C01819=1084.871,371.355,403.473,176.867,26.567,154.395
C01820=1084.877,371.565,403.441,176.870,26.572,154.396
C01821=1084.882,371.775,403.410,176.873,26.578,154.397
C01822=1084.888,372.022,403.373,176.876,26.584,154.398
C01823=1084.894,372.269,403.336,176.880,26.590,154.399
C01824=1084.900,372.516,403.299,176.883,26.596,154.400
C01825=1084.906,372.763,403.262,176.886,26.603,154.401
C01826=1084.913,373.011,403.225,176.890,26.609,154.403
C01827=1084.919,373.257,403.188,176.892,26.615,154.404
C01828=1084.925,373.504,403.151,176.896,26.621,154.405
C01829=1084.932,373.752,403.115,176.900,26.627,154.406
C01830=1084.937,373.998,403.077,176.902,26.633,154.407
C01831=1084.943,374.246,403.040,176.906,26.640,154.408
C01832=1084.949,374.493,403.003,176.909,26.646,154.409
C01833=1084.956,374.740,402.965,176.913,26.652,154.410
C01834=1084.962,374.988,402.928,176.916,26.658,154.412
C01835=1084.968,375.234,402.891,176.919,26.665,154.413
C01836=1084.974,375.481,402.854,176.923,26.672,154.414
C01837=1084.980,375.728,402.816,176.925,26.678,154.415
C01838=1084.986,375.975,402.780,176.929,26.684,154.416
C01839=1084.993,376.223,402.742,176.933,26.690,154.417
C01840=1084.998,376.469,402.704,176.936,26.697,154.418
C01841=1085.004,376.717,402.667,176.939,26.703,154.420
C01842=1085.011,376.963,402.630,176.942,26.709,154.421
C01843=1085.016,377.210,402.593,176.946,26.716,154.422
C01844=1085.023,377.458,402.555,176.948,26.722,154.423
C01845=1085.029,377.705,402.517,176.952,26.729,154.424
C01846=1085.035,377.952,402.480,176.955,26.736,154.426
C01847=1085.041,378.198,402.443,176.959,26.742,154.427
C01848=1085.047,378.446,402.405,176.962,26.748,154.428
C01849=1085.053,378.693,402.367,176.965,26.755,154.429
C01850=1085.060,378.940,402.330,176.969,26.761,154.430
C01851=1085.066,379.187,402.292,176.972,26.768,154.431
C01852=1085.072,379.434,402.255,176.976,26.775,154.433
C01853=1085.078,379.681,402.217,176.979,26.781,154.434
C01854=1085.084,379.928,402.179,176.982,26.788,154.435
C01855=1085.091,380.174,402.141,176.986,26.795,154.436
C01856=1085.097,380.422,402.104,176.989,26.801,154.438
C01857=1085.103,380.669,402.066,176.993,26.808,154.439
C01858=1085.109,380.916,402.029,176.995,26.814,154.440
C01859=1085.115,381.163,401.991,176.999,26.821,154.441
C01860=1085.122,381.410,401.953,177.002,26.828,154.443
C01861=1085.128,381.657,401.916,177.006,26.834,154.444
C01862=1085.135,381.904,401.877,177.009,26.841,154.445
C01863=1085.141,382.151,401.840,177.012,26.847,154.446
C01864=1085.147,382.398,401.802,177.016,26.854,154.447
C01865=1085.153,382.645,401.764,177.019,26.861,154.449
C01866=1085.159,382.891,401.725,177.022,26.868,154.450
C01867=1085.165,383.138,401.688,177.026,26.875,154.451
C01868=1085.172,383.385,401.649,177.030,26.882,154.453
C01869=1085.178,383.632,401.612,177.032,26.888,154.454
C01870=1085.182,383.856,401.577,177.036,26.895,154.455
C01871=1085.188,384.080,401.542,177.038,26.901,154.456
C01872=1085.194,384.304,401.508,177.042,26.908,154.457
C01873=1085.199,384.527,401.473,177.045,26.914,154.459
C01874=1085.205,384.752,401.438,177.047,26.920,154.460
C01875=1085.211,384.975,401.404,177.051,26.926,154.461
C01876=1085.217,385.199,401.369,177.054,26.932,154.462
C01877=1085.222,385.423,401.334,177.057,26.939,154.463
C01878=1085.228,385.671,401.296,177.061,26.946,154.465
C01879=1085.234,385.917,401.258,177.063,26.953,154.466
C01880=1085.241,386.164,401.220,177.067,26.960,154.467
C01881=1085.247,386.410,401.181,177.070,26.967,154.469
C01882=1085.254,386.658,401.143,177.074,26.974,154.470
C01883=1085.260,386.904,401.105,177.077,26.981,154.471
C01884=1085.266,387.152,401.066,177.081,26.988,154.473
C01885=1085.271,387.399,401.028,177.084,26.995,154.474
C01886=1085.278,387.645,400.989,177.088,27.003,154.475
C01887=1085.284,387.891,400.951,177.091,27.010,154.477
C01888=1085.291,388.139,400.913,177.095,27.017,154.478
C01889=1085.296,388.385,400.874,177.098,27.024,154.479
C01890=1085.303,388.633,400.835,177.101,27.031,154.481
C01891=1085.310,388.880,400.797,177.105,27.038,154.482
C01892=1085.316,389.126,400.758,177.108,27.045,154.484
C01893=1085.322,389.373,400.720,177.111,27.053,154.485
C01894=1085.328,389.620,400.681,177.114,27.060,154.486
C01895=1085.335,389.866,400.642,177.118,27.067,154.488
C01896=1085.341,390.114,400.604,177.121,27.075,154.489
C01897=1085.347,390.360,400.566,177.125,27.082,154.491
C01898=1085.354,390.607,400.526,177.128,27.089,154.492
C01899=1085.360,390.854,400.487,177.132,27.096,154.493
C01900=1085.367,391.100,400.449,177.135,27.104,154.495
C01901=1085.372,391.348,400.410,177.139,27.111,154.496
C01902=1085.379,391.595,400.371,177.142,27.119,154.498
C01903=1085.386,391.841,400.332,177.146,27.126,154.499
C01904=1085.391,392.088,400.293,177.149,27.133,154.500
C01905=1085.398,392.335,400.254,177.152,27.141,154.502
C01906=1085.404,392.582,400.215,177.156,27.148,154.503
C01907=1085.411,392.828,400.177,177.159,27.156,154.505
C01908=1085.417,393.075,400.137,177.163,27.163,154.506
C01909=1085.423,393.322,400.098,177.166,27.171,154.508
C01910=1085.429,393.569,400.059,177.170,27.179,154.509
C01911=1085.436,393.815,400.020,177.173,27.186,154.511
C01912=1085.442,394.062,399.981,177.176,27.194,154.512
C01913=1085.449,394.309,399.942,177.180,27.201,154.514
C01914=1085.455,394.556,399.903,177.183,27.209,154.515
C01915=1085.461,394.803,399.864,177.187,27.217,154.517
C01916=1085.467,395.049,399.824,177.191,27.225,154.518
C01917=1085.474,395.296,399.785,177.194,27.232,154.520
C01918=1085.480,395.543,399.746,177.198,27.240,154.521
C01919=1085.486,395.790,399.706,177.201,27.248,154.523
C01920=1085.493,396.037,399.668,177.205,27.256,154.524
C01921=1085.499,396.283,399.627,177.208,27.264,154.526
C01922=1085.505,396.530,399.588,177.211,27.271,154.527
C01923=1085.511,396.777,399.549,177.215,27.279,154.529
C01924=1085.518,397.023,399.509,177.218,27.287,154.530
C01925=1085.524,397.270,399.470,177.222,27.295,154.532
C01926=1085.530,397.501,399.434,177.225,27.302,154.533
C01927=1085.536,397.732,399.396,177.229,27.310,154.535
C01928=1085.542,397.963,399.360,177.231,27.317,154.536
C01929=1085.548,398.194,399.322,177.235,27.325,154.538
C01930=1085.554,398.424,399.285,177.238,27.332,154.539
C01931=1085.560,398.655,399.248,177.242,27.339,154.541
C01932=1085.566,398.886,399.211,177.245,27.347,154.542
C01933=1085.572,399.116,399.174,177.248,27.354,154.544
C01934=1085.578,399.363,399.134,177.252,27.363,154.545
C01935=1085.585,399.610,399.095,177.255,27.371,154.547
C01936=1085.591,399.856,399.055,177.258,27.379,154.549
C01937=1085.597,400.103,399.015,177.262,27.387,154.550
C01938=1085.604,400.350,398.975,177.265,27.395,154.552
C01939=1085.610,400.596,398.935,177.269,27.404,154.553
C01940=1085.616,400.844,398.896,177.272,27.411,154.555
C01941=1085.622,401.090,398.855,177.276,27.420,154.557
C01942=1085.629,401.337,398.815,177.280,27.428,154.558
C01943=1085.635,401.584,398.776,177.283,27.437,154.560
C01944=1085.641,401.830,398.736,177.286,27.445,154.562
C01945=1085.648,402.077,398.695,177.290,27.453,154.563
C01946=1085.655,402.324,398.655,177.294,27.462,154.565
C01947=1085.661,402.571,398.615,177.297,27.470,154.567
C01948=1085.667,402.817,398.575,177.301,27.478,154.568
C01949=1085.673,403.064,398.535,177.304,27.487,154.570
C01950=1085.680,403.311,398.495,177.308,27.495,154.572
C01951=1085.686,403.557,398.455,177.312,27.504,154.573
C01952=1085.693,403.804,398.415,177.315,27.512,154.575
C01953=1085.700,404.051,398.374,177.318,27.521,154.577
C01954=1085.706,404.297,398.334,177.323,27.529,154.579
C01955=1085.712,404.544,398.294,177.326,27.537,154.580
C01956=1085.719,404.790,398.254,177.329,27.546,154.582
C01957=1085.725,405.037,398.214,177.333,27.555,154.584
C01958=1085.731,405.283,398.174,177.337,27.564,154.586
C01959=1085.738,405.531,398.133,177.340,27.572,154.587
C01960=1085.745,405.777,398.092,177.343,27.581,154.589
C01961=1085.751,406.023,398.051,177.348,27.590,154.591
C01962=1085.757,406.270,398.011,177.351,27.598,154.593
C01963=1085.764,406.517,397.971,177.354,27.607,154.594
C01964=1085.771,406.764,397.931,177.359,27.616,154.596
C01965=1085.776,407.010,397.889,177.362,27.625,154.598
C01966=1085.783,407.256,397.849,177.365,27.634,154.600
C01967=1085.790,407.504,397.809,177.369,27.643,154.602
C01968=1085.797,407.750,397.768,177.373,27.652,154.604
C01969=1085.802,407.996,397.727,177.376,27.660,154.605
C01970=1085.809,408.244,397.686,177.380,27.669,154.607
C01971=1085.815,408.490,397.645,177.383,27.679,154.609
C01972=1085.821,408.736,397.605,177.388,27.688,154.611
C01973=1085.828,408.982,397.564,177.391,27.697,154.613
C01974=1085.834,409.230,397.523,177.394,27.705,154.615
C01975=1085.841,409.476,397.482,177.399,27.715,154.616
C01976=1085.847,409.722,397.441,177.402,27.724,154.618
C01977=1085.854,409.969,397.400,177.406,27.733,154.620
C01978=1085.860,410.216,397.360,177.409,27.742,154.622
C01979=1085.867,410.462,397.318,177.413,27.751,154.624
C01980=1085.874,410.708,397.277,177.417,27.761,154.626
C01981=1085.879,410.955,397.236,177.420,27.770,154.628
C01982=1085.886,411.187,397.198,177.424,27.779,154.630
C01983=1085.892,411.418,397.159,177.428,27.788,154.631
C01984=1085.898,411.649,397.121,177.431,27.796,154.633
C01985=1085.904,411.882,397.082,177.434,27.805,154.635
C01986=1085.910,412.113,397.044,177.438,27.814,154.637
C01987=1085.917,412.344,397.004,177.441,27.822,154.639
C01988=1085.923,412.576,396.965,177.444,27.832,154.641
C01989=1085.929,412.807,396.928,177.449,27.841,154.642
C01990=1085.935,413.054,396.886,177.452,27.850,154.644
C01991=1085.942,413.300,396.845,177.456,27.859,154.646
C01992=1085.948,413.547,396.803,177.459,27.869,154.648
C01993=1085.956,413.793,396.762,177.464,27.878,154.650
C01994=1085.962,414.040,396.720,177.467,27.888,154.652
C01995=1085.969,414.286,396.679,177.471,27.897,154.654
C01996=1085.975,414.532,396.638,177.475,27.907,154.656
C01997=1085.982,414.779,396.596,177.479,27.917,154.658
C01998=1085.988,415.025,396.555,177.483,27.926,154.660
C01999=1085.995,415.272,396.513,177.486,27.936,154.662
C02000=1086.002,415.519,396.472,177.490,27.946,154.664
C02001=1086.008,415.765,396.430,177.494,27.956,154.666
C02002=1086.015,416.011,396.389,177.498,27.966,154.668
C02003=1086.022,416.258,396.347,177.502,27.976,154.671
C02004=1086.028,416.504,396.305,177.505,27.985,154.673
C02005=1086.035,416.751,396.263,177.509,27.996,154.675
C02006=1086.041,416.997,396.221,177.513,28.005,154.677
C02007=1086.048,417.243,396.180,177.517,28.016,154.679
C02008=1086.055,417.490,396.138,177.521,28.025,154.681
C02009=1086.061,417.736,396.096,177.525,28.036,154.683
C02010=1086.067,417.983,396.054,177.529,28.046,154.685
C02011=1086.074,418.229,396.012,177.532,28.056,154.687
C02012=1086.080,418.475,395.970,177.536,28.066,154.690
C02013=1086.087,418.721,395.928,177.541,28.076,154.692
C02014=1086.094,418.968,395.886,177.544,28.086,154.694
C02015=1086.101,419.214,395.844,177.548,28.097,154.696
C02016=1086.107,419.460,395.802,177.552,28.107,154.698
C02017=1086.114,419.707,395.760,177.556,28.117,154.700
C02018=1086.121,419.954,395.718,177.560,28.127,154.703
C02019=1086.127,420.200,395.676,177.564,28.138,154.705
C02020=1086.134,420.445,395.633,177.568,28.149,154.707
C02021=1086.140,420.692,395.592,177.572,28.159,154.709
C02022=1086.147,420.939,395.549,177.575,28.169,154.711
C02023=1086.154,421.185,395.506,177.579,28.180,154.714
C02024=1086.162,421.431,395.465,177.583,28.190,154.716
C02025=1086.168,421.677,395.422,177.588,28.201,154.718
C02026=1086.174,421.923,395.381,177.592,28.211,154.720
C02027=1086.181,422.170,395.338,177.596,28.222,154.723
C02028=1086.188,422.416,395.295,177.599,28.233,154.725
C02029=1086.194,422.663,395.252,177.603,28.244,154.727
C02030=1086.201,422.909,395.210,177.607,28.254,154.730
C02031=1086.208,423.155,395.167,177.611,28.265,154.732
C02032=1086.215,423.401,395.125,177.616,28.276,154.734
C02033=1086.221,423.647,395.083,177.620,28.287,154.737
C02034=1086.228,423.893,395.040,177.624,28.298,154.739
C02035=1086.234,424.140,394.997,177.627,28.309,154.741
C02036=1086.241,424.386,394.954,177.631,28.319,154.744
C02037=1086.248,424.632,394.911,177.635,28.331,154.746
C02038=1086.259,425.045,394.840,177.642,28.349,154.750
C02039=1086.271,425.458,394.768,177.649,28.368,154.754
C02040=1086.282,425.871,394.696,177.656,28.386,154.758
C02041=1086.293,426.284,394.624,177.663,28.405,154.762
C02042=1086.300,426.529,394.581,177.667,28.417,154.765
C02043=1086.307,426.775,394.538,177.671,28.428,154.767
C02044=1086.313,427.022,394.495,177.675,28.439,154.769
C02045=1086.320,427.268,394.452,177.679,28.450,154.772
C02046=1086.327,427.514,394.409,177.683,28.462,154.774
C02047=1086.334,427.760,394.366,177.687,28.473,154.777
C02048=1086.341,428.006,394.322,177.691,28.485,154.779
C02049=1086.348,428.253,394.279,177.695,28.496,154.782
C02050=1086.356,428.498,394.236,177.700,28.507,154.784
C02051=1086.362,428.745,394.193,177.704,28.519,154.787
C02052=1086.369,428.991,394.149,177.709,28.531,154.789
C02053=1086.375,429.237,394.106,177.713,28.543,154.792
C02054=1086.382,429.482,394.062,177.717,28.555,154.795
C02055=1086.389,429.729,394.019,177.721,28.566,154.797
C02056=1086.396,429.974,393.976,177.725,28.578,154.800
C02057=1086.403,430.221,393.932,177.729,28.590,154.802
C02058=1086.410,430.467,393.888,177.733,28.602,154.805
C02059=1086.416,430.713,393.845,177.737,28.614,154.808
C02060=1086.423,430.958,393.801,177.741,28.626,154.810
C02061=1086.430,431.204,393.757,177.746,28.638,154.813
C02062=1086.437,431.451,393.713,177.751,28.650,154.815
C02063=1086.444,431.697,393.670,177.755,28.662,154.818
C02064=1086.450,431.943,393.626,177.759,28.674,154.821
C02065=1086.458,432.188,393.583,177.763,28.686,154.823
C02066=1086.465,432.435,393.539,177.767,28.698,154.826
C02067=1086.472,432.681,393.495,177.772,28.710,154.829
C02068=1086.478,432.927,393.452,177.776,28.723,154.832
C02069=1086.485,433.173,393.407,177.780,28.735,154.834
C02070=1086.492,433.419,393.363,177.784,28.748,154.837
C02071=1086.499,433.664,393.320,177.789,28.760,154.840
C02072=1086.506,433.911,393.275,177.793,28.773,154.843
C02073=1086.513,434.156,393.231,177.797,28.785,154.845
C02074=1086.521,434.468,393.175,177.803,28.801,154.849
C02075=1086.530,434.780,393.119,177.808,28.817,154.852
C02076=1086.539,435.092,393.063,177.814,28.833,154.856
C02077=1086.548,435.404,393.007,177.820,28.849,154.860
C02078=1086.555,435.649,392.963,177.824,28.862,154.862
C02079=1086.561,435.895,392.919,177.829,28.875,154.865
C02080=1086.569,436.141,392.874,177.833,28.888,154.868
C02081=1086.575,436.387,392.829,177.837,28.901,154.871
C02082=1086.583,436.633,392.786,177.842,28.914,154.874
C02083=1086.590,436.878,392.741,177.846,28.926,154.877
C02084=1086.597,437.124,392.696,177.850,28.939,154.880
C02085=1086.604,437.370,392.651,177.855,28.953,154.883
C02086=1086.611,437.616,392.607,177.859,28.966,154.886
C02087=1086.618,437.862,392.563,177.864,28.979,154.888
C02088=1086.625,438.108,392.518,177.868,28.992,154.891
C02089=1086.632,438.353,392.473,177.872,29.005,154.894
C02090=1086.639,438.584,392.432,177.876,29.018,154.897
C02091=1086.646,438.814,392.390,177.881,29.030,154.900
C02092=1086.652,439.044,392.347,177.886,29.043,154.903
C02093=1086.658,439.274,392.306,177.890,29.056,154.906
C02094=1086.666,439.505,392.263,177.894,29.068,154.909
C02095=1086.672,439.735,392.222,177.898,29.081,154.911
C02096=1086.679,439.966,392.179,177.902,29.093,154.914
C02097=1086.686,440.196,392.137,177.907,29.106,154.917
C02098=1086.693,440.442,392.092,177.911,29.120,154.920
C02099=1086.700,440.687,392.047,177.916,29.134,154.923
C02100=1086.707,440.933,392.002,177.920,29.147,154.926
C02101=1086.715,441.179,391.957,177.925,29.161,154.930
C02102=1086.721,441.424,391.912,177.930,29.175,154.933
C02103=1086.728,441.670,391.867,177.934,29.189,154.936
C02104=1086.736,441.916,391.821,177.939,29.203,154.939
C02105=1086.743,442.162,391.776,177.943,29.217,154.942
C02106=1086.750,442.407,391.732,177.948,29.231,154.945
C02107=1086.756,442.653,391.685,177.952,29.245,154.949
C02108=1086.764,442.898,391.640,177.957,29.260,154.952
C02109=1086.771,443.144,391.595,177.962,29.274,154.955
C02110=1086.778,443.389,391.549,177.966,29.288,154.958
C02111=1086.785,443.635,391.504,177.971,29.302,154.962
C02112=1086.793,443.881,391.458,177.976,29.317,154.965
C02113=1086.800,444.127,391.412,177.980,29.331,154.968
C02114=1086.807,444.373,391.367,177.985,29.346,154.972
C02115=1086.815,444.618,391.321,177.991,29.360,154.975
C02116=1086.821,444.863,391.276,177.995,29.374,154.978
C02117=1086.829,445.109,391.230,178.000,29.389,154.981
C02118=1086.836,445.354,391.184,178.004,29.404,154.985
C02119=1086.843,445.600,391.138,178.008,29.418,154.988
C02120=1086.851,445.845,391.092,178.012,29.433,154.992
C02121=1086.858,446.091,391.046,178.016,29.448,154.995
C02122=1086.865,446.336,391.001,178.019,29.462,154.999
C02123=1086.872,446.582,390.954,178.022,29.477,155.002
C02124=1086.880,446.828,390.909,178.025,29.491,155.005
C02125=1086.887,447.073,390.862,178.029,29.506,155.009
C02126=1086.894,447.319,390.817,178.032,29.520,155.012
C02127=1086.901,447.565,390.771,178.034,29.535,155.016
C02128=1086.908,447.810,390.724,178.036,29.549,155.019
C02129=1086.916,448.056,390.679,178.038,29.563,155.023
C02130=1086.923,448.301,390.632,178.040,29.578,155.027
C02131=1086.931,448.546,390.586,178.043,29.593,155.030
C02132=1086.938,448.793,390.539,178.044,29.607,155.034
C02133=1086.946,449.038,390.494,178.045,29.621,155.037
C02134=1086.952,449.283,390.447,178.046,29.636,155.041
C02135=1086.960,449.527,390.401,178.048,29.650,155.044
C02136=1086.969,449.773,390.355,178.049,29.664,155.048
C02137=1086.980,450.019,390.311,178.050,29.676,155.051
C02138=1086.604,450.011,390.111,178.013,29.864,155.102
C02139=1086.592,449.765,390.155,178.012,29.851,155.098
C02140=1086.583,449.520,390.202,178.010,29.837,155.095
C02141=1086.576,449.275,390.247,178.009,29.823,155.091
C02142=1086.568,449.031,390.293,178.007,29.808,155.088
C02143=1086.561,448.785,390.339,178.006,29.794,155.084
C02144=1086.554,448.540,390.386,178.005,29.780,155.081
C02145=1086.546,448.294,390.432,178.002,29.765,155.077
C02146=1086.539,448.048,390.479,178.000,29.750,155.074
C02147=1086.531,447.803,390.525,177.998,29.736,155.070
C02148=1086.524,447.557,390.571,177.995,29.721,155.066
C02149=1086.516,447.312,390.617,177.993,29.707,155.063
C02150=1086.510,447.066,390.663,177.990,29.693,155.060
C02151=1086.503,446.820,390.709,177.987,29.678,155.056
C02152=1086.495,446.576,390.756,177.983,29.663,155.053
C02153=1086.488,446.330,390.802,177.980,29.649,155.049
C02154=1086.480,446.084,390.848,177.977,29.634,155.046
C02155=1086.473,445.839,390.894,177.973,29.619,155.042
C02156=1086.466,445.593,390.940,177.969,29.605,155.039
C02157=1086.459,445.347,390.986,177.964,29.590,155.035
C02158=1086.451,445.102,391.031,177.960,29.576,155.032
C02159=1086.443,444.857,391.077,177.955,29.561,155.029
C02160=1086.437,444.611,391.123,177.950,29.546,155.025
C02161=1086.429,444.365,391.168,177.946,29.532,155.022
C02162=1086.422,444.119,391.214,177.941,29.517,155.019
C02163=1086.415,443.874,391.260,177.935,29.503,155.015
C02164=1086.407,443.628,391.306,177.931,29.489,155.012
C02165=1086.401,443.383,391.352,177.926,29.474,155.009
C02166=1086.393,443.137,391.397,177.921,29.460,155.005
C02167=1086.386,442.892,391.442,177.917,29.446,155.002
C02168=1086.378,442.646,391.487,177.912,29.431,154.999
C02169=1086.372,442.400,391.533,177.907,29.417,154.996
C02170=1086.365,442.155,391.579,177.902,29.403,154.993
C02171=1086.357,441.909,391.624,177.897,29.389,154.989
C02172=1086.350,441.664,391.669,177.893,29.375,154.986
C02173=1086.343,441.417,391.715,177.888,29.361,154.983
C02174=1086.336,441.172,391.759,177.884,29.347,154.980
C02175=1086.329,440.927,391.805,177.879,29.333,154.977
C02176=1086.321,440.680,391.850,177.874,29.320,154.974
C02177=1086.314,440.434,391.895,177.869,29.306,154.971
C02178=1086.307,440.190,391.940,177.865,29.292,154.967
C02179=1086.301,439.966,391.982,177.861,29.280,154.965
C02180=1086.294,439.742,392.022,177.857,29.267,154.962
C02181=1086.288,439.519,392.063,177.852,29.255,154.959
C02182=1086.281,439.295,392.104,177.848,29.243,154.956
C02183=1086.275,439.072,392.145,177.844,29.231,154.954
C02184=1086.267,438.849,392.185,177.839,29.218,154.951
C02185=1086.261,438.626,392.226,177.836,29.206,154.948
C02186=1086.255,438.402,392.267,177.832,29.194,154.945
C02187=1086.247,438.156,392.312,177.826,29.181,154.942
C02188=1086.241,437.911,392.356,177.822,29.168,154.939
C02189=1086.233,437.665,392.401,177.818,29.155,154.936
C02190=1086.227,437.420,392.446,177.813,29.141,154.933
C02191=1086.220,437.173,392.490,177.809,29.128,154.931
C02192=1086.212,436.927,392.535,177.804,29.115,154.928
C02193=1086.206,436.681,392.579,177.800,29.102,154.925
C02194=1086.199,436.436,392.624,177.795,29.089,154.922
C02195=1086.191,436.190,392.667,177.790,29.076,154.919
C02196=1086.184,435.944,392.712,177.786,29.063,154.916
C02197=1086.177,435.698,392.757,177.782,29.050,154.913
C02198=1086.171,435.452,392.801,177.777,29.037,154.910
C02199=1086.163,435.206,392.846,177.773,29.025,154.907
C02200=1086.157,434.961,392.890,177.768,29.012,154.905
C02201=1086.150,434.714,392.935,177.764,28.999,154.902
C02202=1086.142,434.469,392.979,177.759,28.987,154.899
C02203=1086.136,434.223,393.022,177.755,28.974,154.896
C02204=1086.129,433.977,393.067,177.751,28.961,154.893
C02205=1086.122,433.731,393.111,177.747,28.949,154.891
C02206=1086.115,433.485,393.155,177.742,28.936,154.888
C02207=1086.107,433.240,393.199,177.738,28.924,154.885
C02208=1086.101,432.994,393.243,177.733,28.912,154.882
C02209=1086.095,432.748,393.287,177.729,28.899,154.880
C02210=1086.088,432.501,393.331,177.725,28.887,154.877
C02211=1086.080,432.255,393.374,177.720,28.875,154.874
C02212=1086.074,432.010,393.419,177.716,28.863,154.872
C02213=1086.066,431.764,393.463,177.712,28.851,154.869
C02214=1086.059,431.518,393.507,177.707,28.838,154.866
C02215=1086.052,431.272,393.550,177.703,28.826,154.863
C02216=1086.045,431.025,393.594,177.699,28.815,154.861
C02217=1086.039,430.779,393.638,177.694,28.802,154.858
C02218=1086.032,430.534,393.681,177.690,28.790,154.856
C02219=1086.025,430.288,393.725,177.686,28.778,154.853
C02220=1086.018,430.042,393.768,177.681,28.766,154.850
C02221=1086.011,429.795,393.812,177.677,28.755,154.848
C02222=1086.004,429.550,393.856,177.673,28.743,154.845
C02223=1085.998,429.303,393.899,177.669,28.731,154.843
C02224=1085.991,429.057,393.942,177.665,28.720,154.840
C02225=1085.984,428.811,393.986,177.661,28.708,154.838
C02226=1085.977,428.566,394.029,177.656,28.696,154.835
C02227=1085.970,428.318,394.073,177.652,28.685,154.832
C02228=1085.963,428.073,394.116,177.648,28.673,154.830
C02229=1085.956,427.827,394.159,177.643,28.661,154.827
C02230=1085.949,427.581,394.202,177.639,28.650,154.825
C02231=1085.943,427.335,394.246,177.634,28.639,154.822
C02232=1085.936,427.089,394.288,177.630,28.627,154.820
C02233=1085.929,426.843,394.331,177.626,28.616,154.817
C02234=1085.922,426.596,394.375,177.622,28.604,154.815
C02235=1085.915,426.356,394.417,177.619,28.593,154.813
C02236=1085.908,426.116,394.458,177.614,28.582,154.810
C02237=1085.902,425.877,394.501,177.610,28.571,154.808
C02238=1085.896,425.636,394.542,177.606,28.561,154.806
C02239=1085.889,425.397,394.585,177.602,28.549,154.803
C02240=1085.882,425.157,394.626,177.598,28.539,154.801
C02241=1085.876,424.917,394.667,177.594,28.528,154.799
C02242=1085.869,424.677,394.710,177.590,28.517,154.796
C02243=1085.862,424.431,394.752,177.586,28.506,154.794
C02244=1085.855,424.184,394.795,177.582,28.495,154.791
C02245=1085.849,423.938,394.837,177.577,28.484,154.789
C02246=1085.842,423.692,394.881,177.574,28.473,154.787
C02247=1085.835,423.446,394.924,177.570,28.462,154.784
C02248=1085.828,423.200,394.966,177.566,28.452,154.782
C02249=1085.822,422.953,395.009,177.562,28.441,154.780
C02250=1085.815,422.707,395.051,177.557,28.430,154.777
C02251=1085.808,422.461,395.094,177.553,28.419,154.775
C02252=1085.802,422.215,395.137,177.549,28.408,154.773
C02253=1085.796,421.969,395.179,177.546,28.398,154.771
C02254=1085.789,421.722,395.222,177.542,28.387,154.768
C02255=1085.781,421.476,395.263,177.537,28.376,154.766
C02256=1085.775,421.229,395.306,177.533,28.366,154.764
C02257=1085.768,420.983,395.348,177.529,28.355,154.761
C02258=1085.761,420.737,395.391,177.526,28.345,154.759
C02259=1085.754,420.491,395.433,177.522,28.334,154.757
C02260=1085.748,420.244,395.475,177.517,28.324,154.755
C02261=1085.741,419.998,395.517,177.513,28.314,154.753
C02262=1085.734,419.752,395.560,177.510,28.303,154.750
C02263=1085.724,419.343,395.630,177.503,28.286,154.747
C02264=1085.712,418.933,395.699,177.497,28.269,154.743
C02265=1085.702,418.525,395.769,177.490,28.252,154.740
C02266=1085.690,418.115,395.839,177.484,28.235,154.736
C02267=1085.684,417.869,395.881,177.479,28.225,154.734
C02268=1085.677,417.623,395.923,177.475,28.215,154.732
C02269=1085.670,417.376,395.965,177.472,28.205,154.730
C02270=1085.664,417.130,396.007,177.467,28.195,154.727
C02271=1085.657,416.884,396.049,177.463,28.184,154.725
C02272=1085.650,416.637,396.090,177.460,28.175,154.723
C02273=1085.644,416.391,396.132,177.456,28.164,154.721
C02274=1085.637,416.144,396.174,177.452,28.154,154.719
C02275=1085.631,415.898,396.216,177.448,28.145,154.717
C02276=1085.624,415.652,396.257,177.444,28.135,154.715
C02277=1085.618,415.405,396.299,177.441,28.125,154.713
C02278=1085.610,415.159,396.341,177.436,28.115,154.711
C02279=1085.604,414.913,396.382,177.432,28.106,154.709
C02280=1085.597,414.666,396.424,177.429,28.096,154.707
C02281=1085.591,414.420,396.465,177.425,28.086,154.705
C02282=1085.584,414.173,396.507,177.421,28.077,154.703
C02283=1085.577,413.926,396.548,177.417,28.067,154.701
C02284=1085.571,413.680,396.590,177.414,28.058,154.699
C02285=1085.564,413.434,396.631,177.409,28.048,154.697
C02286=1085.558,413.187,396.672,177.406,28.039,154.695
C02287=1085.551,412.941,396.714,177.402,28.029,154.693
C02288=1085.545,412.695,396.755,177.399,28.020,154.691
C02289=1085.537,412.448,396.796,177.394,28.010,154.689
C02290=1085.531,412.202,396.838,177.391,28.000,154.687
C02291=1085.523,411.900,396.888,177.386,27.989,154.684
C02292=1085.515,411.598,396.938,177.381,27.978,154.682
C02293=1085.506,411.297,396.989,177.376,27.966,154.680
C02294=1085.500,410.996,397.039,177.372,27.955,154.677
C02295=1085.492,410.749,397.080,177.368,27.945,154.676
C02296=1085.487,410.502,397.121,177.365,27.936,154.674
C02297=1085.479,410.256,397.162,177.360,27.927,154.672
C02298=1085.473,410.010,397.203,177.357,27.918,154.670
C02299=1085.467,409.763,397.244,177.354,27.908,154.668
C02300=1085.460,409.517,397.285,177.349,27.899,154.666
C02301=1085.454,409.270,397.326,177.346,27.890,154.664
C02302=1085.447,409.023,397.367,177.342,27.881,154.662
C02303=1085.440,408.777,397.408,177.339,27.872,154.660
C02304=1085.435,408.530,397.448,177.335,27.863,154.658
C02305=1085.428,408.283,397.489,177.331,27.854,154.657
C02306=1085.422,408.037,397.530,177.328,27.845,154.655
C02307=1085.415,407.790,397.571,177.324,27.836,154.653
C02308=1085.409,407.545,397.611,177.320,27.827,154.651
C02309=1085.402,407.297,397.653,177.317,27.818,154.649
C02310=1085.396,407.051,397.693,177.312,27.809,154.647
C02311=1085.389,406.805,397.734,177.309,27.800,154.646
C02312=1085.382,406.557,397.774,177.306,27.791,154.644
C02313=1085.377,406.311,397.815,177.302,27.782,154.642
C02314=1085.370,406.065,397.856,177.298,27.774,154.640
C02315=1085.364,405.818,397.896,177.295,27.765,154.638
C02316=1085.357,405.571,397.936,177.291,27.756,154.637
C02317=1085.350,405.324,397.976,177.287,27.747,154.635
C02318=1085.345,405.078,398.017,177.284,27.739,154.633
C02319=1085.338,404.831,398.057,177.280,27.730,154.631
C02320=1085.331,404.584,398.098,177.277,27.722,154.630
C02321=1085.325,404.337,398.138,177.272,27.713,154.628
C02322=1085.318,404.091,398.179,177.269,27.704,154.626
C02323=1085.312,403.845,398.219,177.266,27.696,154.624
C02324=1085.305,403.598,398.259,177.262,27.687,154.623
C02325=1085.299,403.352,398.299,177.258,27.679,154.621
C02326=1085.292,403.104,398.339,177.255,27.670,154.619
C02327=1085.286,402.858,398.379,177.251,27.662,154.618
C02328=1085.280,402.611,398.419,177.248,27.654,154.616
C02329=1085.273,402.365,398.460,177.243,27.645,154.614
C02330=1085.267,402.118,398.500,177.240,27.636,154.612
C02331=1085.260,401.872,398.540,177.237,27.628,154.611
C02332=1085.254,401.625,398.580,177.233,27.620,154.609
C02333=1085.247,401.377,398.620,177.230,27.612,154.607
C02334=1085.241,401.131,398.660,177.226,27.604,154.606
C02335=1085.235,400.884,398.700,177.222,27.595,154.604
C02336=1085.228,400.638,398.740,177.219,27.587,154.603
C02337=1085.222,400.390,398.780,177.215,27.579,154.601
C02338=1085.216,400.144,398.820,177.212,27.570,154.599
C02339=1085.209,399.897,398.860,177.208,27.562,154.598
C02340=1085.203,399.651,398.899,177.205,27.554,154.596
C02341=1085.196,399.404,398.939,177.201,27.545,154.594
C02342=1085.190,399.158,398.979,177.197,27.538,154.593
C02343=1085.184,398.926,399.016,177.195,27.530,154.591
C02344=1085.178,398.694,399.053,177.191,27.523,154.590
C02345=1085.172,398.464,399.090,177.188,27.515,154.588
C02346=1085.166,398.233,399.128,177.184,27.508,154.587
C02347=1085.160,398.001,399.165,177.181,27.500,154.585
C02348=1085.154,397.769,399.201,177.178,27.493,154.584
C02349=1085.148,397.538,399.239,177.175,27.485,154.582
C02350=1085.143,397.307,399.276,177.171,27.478,154.581
C02351=1085.136,397.061,399.315,177.168,27.470,154.579
C02352=1085.129,396.814,399.355,177.164,27.462,154.578
C02353=1085.123,396.567,399.394,177.161,27.454,154.576
C02354=1085.117,396.320,399.434,177.157,27.446,154.575
C02355=1085.110,396.074,399.473,177.154,27.438,154.573
C02356=1085.104,395.826,399.513,177.150,27.431,154.572
C02357=1085.098,395.579,399.552,177.147,27.423,154.570
C02358=1085.091,395.333,399.591,177.144,27.415,154.568
C02359=1085.085,395.087,399.631,177.140,27.407,154.567
C02360=1085.079,394.840,399.670,177.137,27.400,154.565
C02361=1085.073,394.593,399.709,177.133,27.392,154.564
C02362=1085.067,394.346,399.749,177.130,27.384,154.562
C02363=1085.060,394.099,399.788,177.126,27.377,154.561
C02364=1085.054,393.852,399.827,177.122,27.368,154.559
C02365=1085.047,393.606,399.865,177.118,27.361,154.558
C02366=1085.041,393.358,399.905,177.115,27.354,154.557
C02367=1085.035,393.112,399.944,177.111,27.346,154.555
C02368=1085.028,392.865,399.984,177.108,27.338,154.554
C02369=1085.022,392.619,400.022,177.105,27.330,154.552
C02370=1085.016,392.372,400.062,177.101,27.323,154.551
C02371=1085.009,392.124,400.100,177.097,27.316,154.549
C02372=1085.004,391.878,400.139,177.095,27.308,154.548
C02373=1084.997,391.631,400.178,177.092,27.301,154.546
C02374=1084.990,391.384,400.217,177.088,27.293,154.545
C02375=1084.984,391.137,400.256,177.085,27.286,154.543
C02376=1084.978,390.891,400.294,177.081,27.279,154.542
C02377=1084.971,390.644,400.333,177.078,27.271,154.540
C02378=1084.965,390.397,400.373,177.074,27.264,154.539
C02379=1084.959,390.150,400.411,177.070,27.257,154.538
C02380=1084.952,389.903,400.449,177.067,27.249,154.536
C02381=1084.946,389.657,400.488,177.064,27.242,154.535
C02382=1084.940,389.410,400.527,177.060,27.235,154.534
C02383=1084.934,389.163,400.565,177.057,27.227,154.532
C02384=1084.927,388.916,400.604,177.053,27.220,154.531
C02385=1084.921,388.670,400.643,177.049,27.213,154.529
C02386=1084.914,388.422,400.681,177.046,27.206,154.528
C02387=1084.908,388.175,400.720,177.042,27.199,154.527
C02388=1084.902,387.929,400.759,177.039,27.191,154.525
C02389=1084.895,387.682,400.797,177.035,27.184,154.524
C02390=1084.889,387.436,400.835,177.032,27.177,154.523
C02391=1084.883,387.188,400.873,177.028,27.170,154.521
C02392=1084.877,386.942,400.912,177.026,27.163,154.520
C02393=1084.871,386.694,400.951,177.022,27.156,154.518
C02394=1084.864,386.448,400.989,177.019,27.149,154.517
C02395=1084.858,386.201,401.027,177.015,27.142,154.516
C02396=1084.851,385.954,401.066,177.012,27.135,154.514
C02397=1084.845,385.707,401.104,177.008,27.128,154.513
C02398=1084.840,385.461,401.143,177.005,27.120,154.512
C02399=1084.834,385.236,401.177,177.002,27.114,154.511
C02400=1084.828,385.012,401.212,176.998,27.108,154.509
C02401=1084.823,384.787,401.247,176.996,27.101,154.508
C02402=1084.816,384.563,401.282,176.993,27.095,154.507
C02403=1084.811,384.337,401.316,176.989,27.089,154.506
C02404=1084.806,384.114,401.351,176.987,27.082,154.505
C02405=1084.800,383.890,401.386,176.983,27.076,154.503
C02406=1084.794,383.665,401.420,176.980,27.070,154.502
C02407=1084.789,383.418,401.459,176.977,27.063,154.501
C02408=1084.782,383.171,401.497,176.973,27.056,154.500
C02409=1084.776,382.924,401.534,176.971,27.049,154.498
C02410=1084.770,382.677,401.572,176.967,27.042,154.497
C02411=1084.764,382.431,401.611,176.963,27.036,154.496
C02412=1084.758,382.184,401.649,176.960,27.029,154.495
C02413=1084.751,381.936,401.687,176.956,27.022,154.493
C02414=1084.745,381.690,401.725,176.953,27.015,154.492
C02415=1084.738,381.442,401.762,176.950,27.009,154.491
C02416=1084.732,381.196,401.800,176.947,27.002,154.489
C02417=1084.726,380.949,401.838,176.943,26.995,154.488
C02418=1084.720,380.702,401.876,176.939,26.988,154.487
C02419=1084.714,380.455,401.914,176.937,26.982,154.486
C02420=1084.707,380.207,401.952,176.933,26.975,154.485
C02421=1084.701,379.961,401.989,176.930,26.969,154.483
C02422=1084.695,379.714,402.026,176.926,26.962,154.482
C02423=1084.689,379.466,402.064,176.923,26.955,154.481
C02424=1084.683,379.219,402.102,176.920,26.949,154.480
C02425=1084.677,378.973,402.140,176.916,26.942,154.479
C02426=1084.670,378.726,402.177,176.913,26.936,154.477
C02427=1084.664,378.479,402.215,176.909,26.929,154.476
C02428=1084.658,378.231,402.252,176.906,26.923,154.475
C02429=1084.652,377.985,402.290,176.903,26.916,154.474
C02430=1084.646,377.737,402.328,176.899,26.909,154.472
C02431=1084.639,377.491,402.365,176.896,26.903,154.471
C02432=1084.633,377.243,402.402,176.893,26.897,154.470
C02433=1084.627,376.997,402.440,176.889,26.890,154.469
C02434=1084.621,376.749,402.478,176.886,26.884,154.468
C02435=1084.615,376.502,402.514,176.883,26.878,154.467
C02436=1084.609,376.255,402.552,176.880,26.871,154.465
C02437=1084.603,376.008,402.589,176.876,26.865,154.464
C02438=1084.596,375.762,402.626,176.872,26.858,154.463
C02439=1084.590,375.514,402.664,176.870,26.852,154.462
C02440=1084.584,375.267,402.701,176.866,26.845,154.461
C02441=1084.578,375.020,402.739,176.863,26.839,154.460
C02442=1084.572,374.773,402.776,176.860,26.833,154.458
C02443=1084.566,374.526,402.813,176.856,26.826,154.457
C02444=1084.561,374.279,402.850,176.853,26.820,154.456
C02445=1084.554,374.031,402.887,176.850,26.814,154.455
C02446=1084.548,373.784,402.925,176.846,26.807,154.454
C02447=1084.541,373.537,402.961,176.843,26.801,154.453
C02448=1084.536,373.290,402.998,176.840,26.795,154.452
C02449=1084.529,373.044,403.036,176.836,26.789,154.450
C02450=1084.524,372.796,403.073,176.833,26.783,154.449
C02451=1084.517,372.548,403.109,176.830,26.776,154.448
C02452=1084.511,372.302,403.147,176.826,26.770,154.447
C02453=1084.504,372.055,403.184,176.823,26.764,154.446
C02454=1084.498,371.808,403.220,176.820,26.758,154.445
C02455=1084.494,371.597,403.252,176.817,26.753,154.444
C02456=1084.488,371.386,403.283,176.814,26.748,154.443
C02457=1084.483,371.176,403.314,176.812,26.742,154.442
C02458=1084.477,370.967,403.346,176.809,26.737,154.441
C02459=1084.471,370.756,403.378,176.806,26.732,154.440
C02460=1084.467,370.546,403.409,176.803,26.727,154.439
C02461=1084.462,370.336,403.440,176.800,26.722,154.438
C02462=1084.456,370.125,403.472,176.797,26.716,154.438
C02463=1084.450,369.878,403.508,176.794,26.710,154.437
C02464=1084.444,369.630,403.545,176.791,26.705,154.435
C02465=1084.438,369.383,403.582,176.787,26.699,154.434
C02466=1084.432,369.136,403.618,176.785,26.692,154.433
C02467=1084.426,368.889,403.655,176.781,26.686,154.432
C02468=1084.420,368.642,403.692,176.777,26.680,154.431
C02469=1084.414,368.395,403.729,176.775,26.674,154.430
C02470=1084.408,368.148,403.765,176.771,26.668,154.429
C02471=1084.401,367.900,403.802,176.768,26.663,154.428
C02472=1084.396,367.653,403.839,176.764,26.657,154.427
C02473=1084.389,367.406,403.875,176.761,26.651,154.426
C02474=1084.383,367.158,403.911,176.758,26.645,154.425
C02475=1084.378,366.911,403.948,176.754,26.639,154.424
C02476=1084.371,366.664,403.984,176.752,26.633,154.423
C02477=1084.365,366.417,404.021,176.748,26.627,154.422
C02478=1084.359,366.171,404.057,176.745,26.621,154.421
C02479=1084.354,365.923,404.093,176.742,26.615,154.420
C02480=1084.348,365.676,404.129,176.738,26.609,154.419
C02481=1084.341,365.428,404.166,176.735,26.603,154.418
C02482=1084.335,365.181,404.202,176.732,26.598,154.417
C02483=1084.330,364.933,404.239,176.729,26.592,154.416
C02484=1084.323,364.686,404.275,176.725,26.586,154.415
C02485=1084.317,364.439,404.312,176.722,26.581,154.414
C02486=1084.311,364.192,404.347,176.719,26.575,154.413
C02487=1084.305,363.945,404.384,176.716,26.569,154.412
C02488=1084.299,363.697,404.420,176.712,26.563,154.411
C02489=1084.292,363.450,404.456,176.709,26.557,154.410
C02490=1084.287,363.204,404.492,176.706,26.552,154.409
C02491=1084.281,362.956,404.528,176.702,26.546,154.408
C02492=1084.274,362.709,404.564,176.699,26.541,154.407
C02493=1084.268,362.461,404.600,176.696,26.535,154.406
C02494=1084.262,362.214,404.636,176.693,26.529,154.405
C02495=1084.257,361.966,404.673,176.689,26.523,154.404
C02496=1084.250,361.719,404.709,176.686,26.518,154.403
C02497=1084.244,361.471,404.745,176.683,26.512,154.402
C02498=1084.239,361.224,404.780,176.680,26.507,154.401
C02499=1084.232,360.977,404.817,176.676,26.501,154.400
C02500=1084.226,360.730,404.852,176.673,26.496,154.399
C02501=1084.220,360.482,404.888,176.670,26.490,154.398
C02502=1084.214,360.235,404.925,176.667,26.484,154.397
C02503=1084.209,359.988,404.960,176.663,26.479,154.396
C02504=1084.202,359.741,404.995,176.661,26.473,154.395
C02505=1084.196,359.494,405.032,176.657,26.467,154.394
C02506=1084.190,359.246,405.067,176.654,26.462,154.393
C02507=1084.183,358.998,405.103,176.650,26.457,154.392
C02508=1084.178,358.751,405.138,176.648,26.451,154.391
C02509=1084.172,358.504,405.174,176.644,26.446,154.391
C02510=1084.166,358.256,405.211,176.641,26.440,154.390
C02511=1084.156,357.852,405.268,176.636,26.432,154.388
C02512=1084.146,357.447,405.327,176.630,26.422,154.387
C02513=1084.136,357.042,405.385,176.625,26.413,154.385
C02514=1084.126,356.638,405.443,176.620,26.405,154.384
C02515=1084.120,356.390,405.479,176.616,26.399,154.383
C02516=1084.114,356.143,405.515,176.614,26.394,154.382
C02517=1084.108,355.896,405.549,176.611,26.389,154.381
C02518=1084.102,355.648,405.585,176.607,26.383,154.380
C02519=1084.096,355.400,405.620,176.604,26.378,154.379
C02520=1084.091,355.153,405.655,176.601,26.372,154.378
C02521=1084.085,354.905,405.691,176.598,26.367,154.377
C02522=1084.078,354.658,405.726,176.594,26.361,154.376
C02523=1084.072,354.411,405.762,176.591,26.357,154.376
C02524=1084.066,354.163,405.797,176.588,26.351,154.375
C02525=1084.060,353.916,405.832,176.585,26.346,154.374
C02526=1084.054,353.669,405.868,176.582,26.340,154.373
C02527=1084.048,353.421,405.903,176.578,26.335,154.372
C02528=1084.042,353.173,405.939,176.575,26.330,154.371
C02529=1084.036,352.926,405.973,176.572,26.325,154.370
C02530=1084.030,352.679,406.009,176.569,26.320,154.369
C02531=1084.024,352.431,406.043,176.566,26.314,154.368
C02532=1084.018,352.184,406.079,176.562,26.309,154.368
C02533=1084.012,351.936,406.115,176.559,26.304,154.367
C02534=1084.006,351.689,406.149,176.556,26.299,154.366
C02535=1084.000,351.441,406.184,176.553,26.293,154.365
C02536=1083.994,351.194,406.219,176.550,26.289,154.364
C02537=1083.988,350.946,406.254,176.546,26.283,154.363
C02538=1083.982,350.699,406.289,176.543,26.278,154.363
C02539=1083.976,350.452,406.325,176.540,26.273,154.362
C02540=1083.970,350.204,406.359,176.537,26.268,154.361
C02541=1083.964,349.957,406.394,176.534,26.262,154.360
C02542=1083.958,349.709,406.429,176.531,26.258,154.359
C02543=1083.953,349.462,406.464,176.527,26.252,154.358
C02544=1083.946,349.214,406.499,176.524,26.247,154.357
C02545=1083.941,348.967,406.534,176.522,26.242,154.357
C02546=1083.934,348.719,406.568,176.518,26.237,154.356
C02547=1083.929,348.472,406.604,176.515,26.232,154.355
C02548=1083.922,348.224,406.638,176.512,26.227,154.354
C02549=1083.916,347.977,406.673,176.508,26.222,154.353
C02550=1083.910,347.729,406.708,176.505,26.217,154.353
C02551=1083.905,347.482,406.742,176.503,26.212,154.352
C02552=1083.898,347.234,406.778,176.499,26.207,154.351
C02553=1083.893,346.987,406.812,176.496,26.202,154.350
C02554=1083.886,346.739,406.846,176.493,26.197,154.349
C02555=1083.881,346.492,406.882,176.489,26.192,154.349
C02556=1083.874,346.244,406.916,176.487,26.187,154.348
C02557=1083.869,345.996,406.951,176.484,26.182,154.347
C02558=1083.863,345.749,406.985,176.480,26.177,154.346
C02559=1083.857,345.502,407.020,176.477,26.172,154.345
C02560=1083.851,345.254,407.055,176.474,26.167,154.344
C02561=1083.845,345.006,407.089,176.470,26.162,154.344
C02562=1083.839,344.759,407.123,176.467,26.157,154.343
C02563=1083.830,344.357,407.179,176.462,26.149,154.342
C02564=1083.819,343.955,407.235,176.457,26.141,154.340
C02565=1083.810,343.553,407.291,176.452,26.133,154.339
C02566=1083.801,343.151,407.346,176.447,26.125,154.338
C02567=1083.794,342.903,407.381,176.444,26.120,154.337
C02568=1083.788,342.656,407.415,176.441,26.115,154.336
C02569=1083.782,342.409,407.449,176.437,26.110,154.335
C02570=1083.777,342.160,407.484,176.434,26.106,154.335
C02571=1083.771,341.913,407.518,176.432,26.101,154.334
C02572=1083.765,341.666,407.552,176.429,26.096,154.333
C02573=1083.759,341.418,407.586,176.425,26.091,154.332
C02574=1083.753,341.171,407.620,176.422,26.086,154.332
C02575=1083.747,340.923,407.655,176.419,26.082,154.331
C02576=1083.740,340.675,407.689,176.416,26.077,154.330
C02577=1083.735,340.428,407.723,176.413,26.072,154.329
C02578=1083.729,340.181,407.757,176.410,26.067,154.329
C02579=1083.723,339.932,407.791,176.407,26.063,154.328
C02580=1083.717,339.685,407.825,176.404,26.058,154.327
C02581=1083.712,339.437,407.859,176.400,26.053,154.326
C02582=1083.706,339.190,407.894,176.397,26.048,154.326
C02583=1083.699,338.942,407.928,176.394,26.043,154.325
C02584=1083.694,338.694,407.961,176.391,26.039,154.324
C02585=1083.688,338.447,407.995,176.388,26.034,154.324
C02586=1083.682,338.200,408.029,176.385,26.029,154.323
C02587=1083.676,337.951,408.063,176.382,26.024,154.322
C02588=1083.670,337.704,408.097,176.379,26.020,154.321
C02589=1083.664,337.456,408.131,176.376,26.015,154.320
C02590=1083.658,337.209,408.165,176.372,26.010,154.320
C02591=1083.652,336.961,408.199,176.369,26.005,154.319
C02592=1083.646,336.713,408.233,176.366,26.001,154.318
C02593=1083.640,336.466,408.266,176.363,25.997,154.318
C02594=1083.634,336.218,408.300,176.361,25.992,154.317
C02595=1083.628,335.970,408.333,176.357,25.987,154.316
C02596=1083.622,335.722,408.368,176.354,25.982,154.315
C02597=1083.616,335.475,408.401,176.351,25.978,154.315
C02598=1083.611,335.227,408.435,176.348,25.973,154.314
C02599=1083.605,334.979,408.468,176.345,25.969,154.313
C02600=1083.598,334.732,408.502,176.341,25.964,154.313
C02601=1083.593,334.485,408.535,176.338,25.959,154.312
C02602=1083.586,334.237,408.570,176.335,25.955,154.311
C02603=1083.581,333.989,408.603,176.332,25.950,154.311
C02604=1083.575,333.741,408.637,176.330,25.946,154.310
C02605=1083.569,333.493,408.670,176.327,25.941,154.309
C02606=1083.563,333.246,408.703,176.323,25.936,154.309
C02607=1083.557,332.999,408.737,176.320,25.932,154.308
C02608=1083.552,332.751,408.770,176.317,25.927,154.307
C02609=1083.546,332.503,408.804,176.314,25.923,154.306
C02610=1083.540,332.255,408.838,176.311,25.918,154.306
C02611=1083.534,332.008,408.871,176.308,25.914,154.305
C02612=1083.528,331.759,408.904,176.304,25.909,154.304
C02613=1083.522,331.511,408.938,176.301,25.905,154.304
C02614=1083.516,331.264,408.971,176.298,25.900,154.303
C02615=1083.506,330.857,409.025,176.293,25.893,154.302
C02616=1083.496,330.449,409.081,176.289,25.886,154.301
C02617=1083.486,330.042,409.135,176.284,25.878,154.300
C02618=1083.477,329.634,409.189,176.278,25.871,154.299
C02619=1083.470,329.387,409.223,176.276,25.867,154.298
C02620=1083.464,329.139,409.256,176.273,25.862,154.297
C02621=1083.458,328.891,409.289,176.270,25.858,154.297
C02622=1083.452,328.644,409.322,176.267,25.854,154.296
C02623=1083.447,328.396,409.355,176.263,25.849,154.295
C02624=1083.440,328.148,409.388,176.260,25.845,154.295
C02625=1083.435,327.900,409.421,176.257,25.840,154.294
C02626=1083.428,327.653,409.454,176.254,25.836,154.293
C02627=1083.423,327.405,409.487,176.251,25.832,154.293
C02628=1083.417,327.157,409.520,176.248,25.827,154.292
C02629=1083.411,326.909,409.553,176.245,25.823,154.291
C02630=1083.405,326.662,409.586,176.242,25.818,154.291
C02631=1083.398,326.414,409.619,176.239,25.815,154.290
C02632=1083.393,326.166,409.651,176.236,25.810,154.290
C02633=1083.387,325.918,409.684,176.232,25.805,154.289
C02634=1083.381,325.670,409.717,176.229,25.801,154.288
C02635=1083.375,325.422,409.750,176.226,25.797,154.288
C02636=1083.369,325.175,409.783,176.223,25.792,154.287
C02637=1083.363,324.927,409.816,176.220,25.788,154.286
C02638=1083.357,324.679,409.848,176.217,25.784,154.286
C02639=1083.352,324.431,409.882,176.215,25.780,154.285
C02640=1083.345,324.183,409.914,176.212,25.775,154.284
C02641=1083.339,323.936,409.947,176.209,25.771,154.284
C02642=1083.334,323.687,409.980,176.206,25.767,154.283
C02643=1083.328,323.440,410.012,176.203,25.763,154.283
C02644=1083.322,323.193,410.045,176.200,25.758,154.282
C02645=1083.316,322.945,410.078,176.197,25.754,154.281
C02646=1083.310,322.697,410.110,176.194,25.749,154.281
C02647=1083.304,322.449,410.143,176.191,25.746,154.280
C02648=1083.298,322.201,410.176,176.188,25.741,154.279
C02649=1083.293,321.954,410.208,176.184,25.736,154.279
C02650=1083.287,321.706,410.241,176.181,25.732,154.278
C02651=1083.281,321.457,410.273,176.178,25.728,154.278
C02652=1083.275,321.210,410.306,176.175,25.724,154.277
C02653=1083.269,320.962,410.339,176.172,25.719,154.276
C02654=1083.264,320.714,410.371,176.169,25.715,154.276
C02655=1083.258,320.467,410.404,176.166,25.711,154.275
C02656=1083.252,320.219,410.436,176.163,25.707,154.274
C02657=1083.246,319.971,410.469,176.160,25.703,154.274
C02658=1083.240,319.722,410.501,176.157,25.698,154.273
C02659=1083.235,319.476,410.534,176.155,25.694,154.273
C02660=1083.229,319.227,410.566,176.151,25.690,154.272
C02661=1083.223,318.979,410.598,176.149,25.686,154.271
C02662=1083.218,318.732,410.631,176.146,25.681,154.271
C02663=1083.212,318.484,410.663,176.143,25.677,154.270
C02664=1083.206,318.236,410.695,176.140,25.673,154.269
C02665=1083.200,317.988,410.728,176.137,25.668,154.269
C02666=1083.195,317.740,410.760,176.134,25.665,154.268
C02667=1083.186,317.326,410.814,176.129,25.657,154.267
C02668=1083.175,316.912,410.868,176.124,25.650,154.266
C02669=1083.166,316.498,410.921,176.119,25.643,154.265
C02670=1083.156,316.084,410.976,176.115,25.636,154.264
C02671=1083.151,315.836,411.008,176.112,25.632,154.264
C02672=1083.145,315.588,411.039,176.109,25.628,154.263
C02673=1083.139,315.340,411.071,176.106,25.624,154.262
C02674=1083.134,315.092,411.105,176.103,25.620,154.262
C02675=1083.128,314.845,411.136,176.100,25.616,154.261
C02676=1083.122,314.596,411.168,176.097,25.611,154.261
C02677=1083.115,314.348,411.200,176.094,25.607,154.260
C02678=1083.110,314.101,411.231,176.091,25.604,154.259
C02679=1083.104,313.853,411.263,176.088,25.600,154.259
C02680=1083.098,313.604,411.295,176.085,25.595,154.258
C02681=1083.092,313.356,411.327,176.082,25.591,154.258
C02682=1083.086,313.110,411.359,176.079,25.587,154.257
C02683=1083.080,312.861,411.391,176.076,25.583,154.257
C02684=1083.074,312.613,411.423,176.073,25.580,154.256
C02685=1083.068,312.366,411.455,176.070,25.575,154.256
C02686=1083.062,312.118,411.486,176.067,25.571,154.255
C02687=1083.056,311.870,411.518,176.064,25.567,154.254
C02688=1083.050,311.622,411.550,176.061,25.563,154.254
C02689=1083.044,311.374,411.582,176.058,25.559,154.253
C02690=1083.038,311.127,411.613,176.055,25.556,154.253
C02691=1083.032,310.878,411.644,176.052,25.551,154.252
C02692=1083.027,310.630,411.676,176.049,25.547,154.252
C02693=1083.021,310.382,411.708,176.046,25.543,154.251
C02694=1083.014,310.134,411.740,176.043,25.539,154.251
C02695=1083.009,309.887,411.771,176.040,25.535,154.250
C02696=1083.003,309.639,411.803,176.038,25.532,154.250
C02697=1082.997,309.391,411.834,176.034,25.528,154.249
C02698=1082.991,309.143,411.866,176.032,25.523,154.248
C02699=1082.986,308.895,411.897,176.029,25.520,154.248
C02700=1082.980,308.647,411.929,176.026,25.516,154.247
C02701=1082.974,308.400,411.960,176.023,25.512,154.247
C02702=1082.968,308.151,411.992,176.019,25.508,154.246
C02703=1082.963,307.903,412.023,176.016,25.504,154.246
C02704=1082.956,307.655,412.055,176.013,25.500,154.245
C02705=1082.951,307.408,412.087,176.010,25.496,154.245
C02706=1082.944,307.160,412.118,176.007,25.492,154.244
C02707=1082.939,306.912,412.149,176.005,25.488,154.243
C02708=1082.933,306.664,412.181,176.001,25.484,154.243
C02709=1082.927,306.416,412.212,175.999,25.480,154.242
C02710=1082.922,306.168,412.243,175.996,25.476,154.242
C02711=1082.916,305.920,412.275,175.993,25.472,154.241
C02712=1082.910,305.672,412.305,175.990,25.468,154.241
C02713=1082.904,305.424,412.337,175.987,25.464,154.240
C02714=1082.898,305.177,412.368,175.984,25.460,154.240
C02715=1082.893,304.929,412.399,175.981,25.456,154.239
C02716=1082.887,304.680,412.431,175.978,25.453,154.239
C02717=1082.881,304.433,412.462,175.975,25.449,154.238
C02718=1082.875,304.185,412.493,175.972,25.445,154.238
C02719=1082.865,303.774,412.545,175.968,25.438,154.237
C02720=1082.856,303.363,412.597,175.963,25.431,154.236
C02721=1082.846,302.951,412.649,175.958,25.425,154.235
C02722=1082.837,302.540,412.700,175.954,25.419,154.234
C02723=1082.831,302.292,412.731,175.951,25.415,154.233
C02724=1082.826,302.044,412.762,175.948,25.411,154.233
C02725=1082.820,301.796,412.794,175.945,25.407,154.232
C02726=1082.814,301.548,412.824,175.942,25.403,154.232
C02727=1082.809,301.300,412.855,175.939,25.399,154.231
C02728=1082.803,301.053,412.886,175.936,25.395,154.231
C02729=1082.797,300.804,412.918,175.934,25.391,154.230
C02730=1082.791,300.556,412.948,175.931,25.387,154.230
C02731=1082.786,300.308,412.979,175.928,25.383,154.229
C02732=1082.780,300.061,413.010,175.925,25.380,154.229
C02733=1082.774,299.812,413.041,175.922,25.376,154.228
C02734=1082.768,299.564,413.072,175.919,25.372,154.228
C02735=1082.763,299.316,413.103,175.916,25.368,154.227
C02736=1082.757,299.069,413.134,175.914,25.364,154.227
C02737=1082.752,298.821,413.165,175.911,25.360,154.226
C02738=1082.746,298.572,413.195,175.908,25.356,154.226
C02739=1082.741,298.324,413.226,175.905,25.352,154.225
C02740=1082.735,298.076,413.257,175.902,25.348,154.224
C02741=1082.729,297.829,413.288,175.899,25.344,154.224
C02742=1082.724,297.581,413.319,175.896,25.341,154.223
C02743=1082.717,297.332,413.349,175.893,25.337,154.223
C02744=1082.711,297.085,413.380,175.890,25.333,154.222
C02745=1082.706,296.837,413.410,175.887,25.329,154.222
C02746=1082.701,296.589,413.441,175.884,25.325,154.221
C02747=1082.694,296.340,413.472,175.881,25.322,154.221
C02748=1082.688,296.092,413.502,175.879,25.318,154.220
C02749=1082.682,295.844,413.532,175.876,25.314,154.220
C02750=1082.677,295.597,413.563,175.873,25.310,154.219
C02751=1082.672,295.348,413.594,175.870,25.307,154.219
C02752=1082.665,295.100,413.624,175.867,25.303,154.218
C02753=1082.659,294.852,413.655,175.864,25.299,154.218
C02754=1082.654,294.604,413.685,175.862,25.295,154.217
C02755=1082.648,294.356,413.715,175.859,25.292,154.217
C02756=1082.642,294.109,413.746,175.856,25.288,154.216
C02757=1082.636,293.860,413.775,175.853,25.284,154.216
C02758=1082.631,293.611,413.807,175.850,25.281,154.216
C02759=1082.625,293.364,413.837,175.848,25.277,154.215
C02760=1082.619,293.116,413.867,175.845,25.273,154.214
C02761=1082.613,292.868,413.898,175.842,25.269,154.214
C02762=1082.607,292.620,413.928,175.838,25.266,154.214
C02763=1082.602,292.372,413.958,175.835,25.262,154.213
C02764=1082.596,292.124,413.988,175.833,25.258,154.212
C02765=1082.590,291.876,414.018,175.830,25.255,154.212
C02766=1082.584,291.627,414.049,175.827,25.251,154.212
C02767=1082.578,291.380,414.080,175.824,25.247,154.211
C02768=1082.573,291.131,414.109,175.822,25.244,154.211
C02769=1082.567,290.883,414.140,175.819,25.240,154.210
C02770=1082.561,290.636,414.170,175.816,25.236,154.210
C02771=1082.552,290.238,414.219,175.812,25.230,154.209
C02772=1082.543,289.842,414.266,175.807,25.224,154.208
C02773=1082.534,289.444,414.314,175.803,25.218,154.207
C02774=1082.524,289.047,414.362,175.798,25.212,154.207
C02775=1082.519,288.799,414.393,175.795,25.208,154.206
C02776=1082.513,288.551,414.423,175.792,25.205,154.206
C02777=1082.507,288.303,414.453,175.790,25.201,154.205
C02778=1082.501,288.055,414.482,175.787,25.198,154.205
C02779=1082.495,287.807,414.512,175.784,25.194,154.204
C02780=1082.489,287.559,414.542,175.781,25.190,154.204
C02781=1082.484,287.311,414.572,175.779,25.187,154.203
C02782=1082.478,287.063,414.602,175.775,25.183,154.203
C02783=1082.473,286.815,414.632,175.772,25.179,154.202
C02784=1082.466,286.567,414.662,175.769,25.176,154.202
C02785=1082.461,286.319,414.691,175.767,25.172,154.201
C02786=1082.455,286.070,414.721,175.764,25.169,154.201
C02787=1082.449,285.822,414.751,175.761,25.165,154.200
C02788=1082.444,285.574,414.781,175.758,25.161,154.200
C02789=1082.437,285.326,414.811,175.756,25.158,154.200
C02790=1082.432,285.078,414.840,175.753,25.154,154.199
C02791=1082.426,284.829,414.870,175.750,25.150,154.199
C02792=1082.420,284.582,414.900,175.747,25.146,154.198
C02793=1082.415,284.333,414.930,175.745,25.143,154.198
C02794=1082.409,284.085,414.959,175.742,25.139,154.197
C02795=1082.403,283.837,414.989,175.739,25.136,154.197
C02796=1082.397,283.589,415.019,175.737,25.132,154.196
C02797=1082.392,283.340,415.049,175.733,25.129,154.196
C02798=1082.385,283.092,415.078,175.731,25.125,154.195
C02799=1082.380,282.844,415.107,175.727,25.121,154.195
C02800=1082.374,282.596,415.138,175.725,25.118,154.194
C02801=1082.369,282.348,415.167,175.722,25.114,154.194
C02802=1082.363,282.100,415.196,175.719,25.110,154.193
C02803=1082.357,281.852,415.226,175.717,25.107,154.193
C02804=1082.352,281.603,415.255,175.714,25.103,154.192
C02805=1082.345,281.356,415.285,175.711,25.099,154.192
C02806=1082.340,281.107,415.315,175.708,25.095,154.192
C02807=1082.334,280.859,415.344,175.706,25.092,154.191
C02808=1082.328,280.611,415.373,175.703,25.089,154.191
C02809=1082.323,280.362,415.403,175.700,25.085,154.190
C02810=1082.318,280.114,415.432,175.698,25.082,154.190
C02811=1082.311,279.866,415.461,175.695,25.078,154.189
C02812=1082.306,279.618,415.491,175.691,25.074,154.189
C02813=1082.300,279.370,415.520,175.689,25.071,154.188
C02814=1082.294,279.121,415.549,175.686,25.067,154.188
C02815=1082.288,278.873,415.579,175.683,25.064,154.188
C02816=1082.282,278.625,415.608,175.681,25.061,154.187
C02817=1082.277,278.377,415.637,175.678,25.057,154.187
C02818=1082.271,278.129,415.666,175.675,25.053,154.186
C02819=1082.265,277.881,415.696,175.672,25.049,154.186
C02820=1082.259,277.632,415.725,175.670,25.046,154.185
C02821=1082.253,277.384,415.754,175.667,25.042,154.185
C02822=1082.248,277.136,415.784,175.664,25.038,154.184
C02823=1082.239,276.749,415.829,175.660,25.033,154.184
C02824=1082.230,276.361,415.874,175.656,25.028,154.183
C02825=1082.221,275.973,415.920,175.651,25.022,154.182
C02826=1082.212,275.587,415.965,175.647,25.017,154.182
C02827=1082.207,275.338,415.994,175.644,25.013,154.181
C02828=1082.200,275.090,416.023,175.641,25.009,154.181
C02829=1082.195,274.842,416.052,175.639,25.006,154.180
C02830=1082.189,274.594,416.081,175.636,25.003,154.180
C02831=1082.184,274.345,416.110,175.633,24.999,154.179
C02832=1082.178,274.097,416.139,175.631,24.996,154.179
C02833=1082.172,273.850,416.168,175.628,24.992,154.179
C02834=1082.167,273.601,416.197,175.625,24.988,154.178
C02835=1082.161,273.352,416.226,175.623,24.985,154.178
C02836=1082.154,273.104,416.255,175.620,24.981,154.177
C02837=1082.150,272.856,416.283,175.616,24.978,154.177
C02838=1082.143,272.608,416.312,175.614,24.974,154.176
C02839=1082.137,272.360,416.341,175.611,24.971,154.176
C02840=1082.131,272.111,416.370,175.608,24.967,154.176
C02841=1082.126,271.863,416.399,175.606,24.964,154.175
C02842=1082.120,271.614,416.427,175.603,24.960,154.175
C02843=1082.114,271.366,416.456,175.601,24.957,154.174
C02844=1082.109,271.119,416.485,175.598,24.953,154.174
C02845=1082.103,270.870,416.514,175.595,24.949,154.173
C02846=1082.097,270.622,416.543,175.593,24.946,154.173
C02847=1082.092,270.374,416.571,175.590,24.943,154.172
C02848=1082.085,270.126,416.600,175.587,24.939,154.172
C02849=1082.080,269.876,416.629,175.585,24.936,154.171
C02850=1082.075,269.629,416.658,175.581,24.932,154.171
C02851=1082.069,269.380,416.686,175.579,24.929,154.171
C02852=1082.063,269.132,416.714,175.576,24.926,154.170
C02853=1082.057,268.884,416.743,175.573,24.922,154.170
C02854=1082.051,268.635,416.771,175.571,24.918,154.169
C02855=1082.046,268.387,416.801,175.568,24.915,154.169
C02856=1082.040,268.139,416.829,175.565,24.911,154.169
C02857=1082.034,267.890,416.857,175.563,24.908,154.168
C02858=1082.029,267.643,416.886,175.560,24.904,154.168
C02859=1082.023,267.394,416.914,175.558,24.901,154.167
C02860=1082.017,267.145,416.942,175.554,24.898,154.167
C02861=1082.011,266.898,416.971,175.551,24.894,154.166
C02862=1082.005,266.649,416.999,175.549,24.891,154.166
C02863=1082.000,266.401,417.027,175.546,24.887,154.166
C02864=1081.994,266.152,417.056,175.544,24.884,154.165
C02865=1081.988,265.904,417.085,175.541,24.880,154.165
C02866=1081.982,265.656,417.113,175.538,24.877,154.164
C02867=1081.977,265.407,417.142,175.536,24.873,154.164
C02868=1081.972,265.159,417.170,175.533,24.870,154.163
C02869=1081.966,264.911,417.199,175.531,24.866,154.163
C02870=1081.960,264.663,417.227,175.528,24.863,154.163
C02871=1081.954,264.414,417.255,175.525,24.860,154.162
C02872=1081.949,264.166,417.283,175.522,24.856,154.162
C02873=1081.943,263.917,417.311,175.519,24.852,154.161
C02874=1081.936,263.669,417.339,175.517,24.849,154.161
C02875=1081.927,263.284,417.383,175.513,24.844,154.160
C02876=1081.918,262.900,417.426,175.509,24.839,154.160
C02877=1081.910,262.517,417.470,175.504,24.834,154.159
C02878=1081.900,262.132,417.513,175.501,24.828,154.158
C02879=1081.894,261.883,417.541,175.498,24.825,154.158
C02880=1081.889,261.635,417.569,175.495,24.821,154.158
C02881=1081.883,261.386,417.597,175.492,24.818,154.157
C02882=1081.877,261.139,417.625,175.489,24.815,154.157
C02883=1081.871,260.890,417.653,175.487,24.811,154.156
C02884=1081.865,260.641,417.681,175.484,24.808,154.156
C02885=1081.860,260.393,417.709,175.482,24.805,154.156
C02886=1081.853,260.145,417.737,175.479,24.801,154.155
C02887=1081.848,259.897,417.765,175.477,24.798,154.155
C02888=1081.842,259.648,417.793,175.474,24.795,154.154
C02889=1081.837,259.400,417.821,175.471,24.791,154.154
C02890=1081.830,259.151,417.849,175.468,24.788,154.154
C02891=1081.825,258.903,417.876,175.465,24.784,154.153
C02892=1081.819,258.655,417.904,175.463,24.781,154.153
C02893=1081.813,258.406,417.932,175.460,24.777,154.152
C02894=1081.807,258.158,417.960,175.458,24.774,154.152
C02895=1081.802,257.909,417.988,175.455,24.771,154.151
C02896=1081.796,257.661,418.015,175.453,24.767,154.151
C02897=1081.790,257.412,418.043,175.450,24.764,154.151
C02898=1081.784,257.164,418.071,175.448,24.761,154.150
C02899=1081.779,256.915,418.099,175.445,24.757,154.150
C02900=1081.773,256.667,418.126,175.441,24.754,154.149
C02901=1081.767,256.419,418.154,175.439,24.751,154.149
C02902=1081.761,256.170,418.182,175.436,24.747,154.149
C02903=1081.755,255.923,418.210,175.434,24.744,154.148
C02904=1081.750,255.674,418.237,175.431,24.740,154.148
C02905=1081.744,255.425,418.265,175.429,24.737,154.147
C02906=1081.738,255.177,418.293,175.426,24.733,154.147
C02907=1081.733,254.928,418.320,175.424,24.730,154.147
C02908=1081.727,254.680,418.348,175.421,24.726,154.146
C02909=1081.722,254.432,418.375,175.419,24.723,154.146
C02910=1081.716,254.183,418.403,175.415,24.720,154.145
C02911=1081.710,253.935,418.431,175.413,24.717,154.145
C02912=1081.705,253.686,418.458,175.410,24.713,154.145
C02913=1081.699,253.438,418.486,175.408,24.710,154.144
C02914=1081.693,253.189,418.513,175.405,24.706,154.144
C02915=1081.687,252.941,418.541,175.403,24.703,154.143
C02916=1081.682,252.693,418.567,175.400,24.699,154.143
C02917=1081.676,252.444,418.596,175.398,24.696,154.142
C02918=1081.671,252.196,418.623,175.395,24.692,154.142
C02919=1081.665,251.948,418.650,175.393,24.689,154.142
C02920=1081.659,251.698,418.678,175.390,24.686,154.141
C02921=1081.653,251.451,418.705,175.387,24.683,154.141
C02922=1081.648,251.202,418.733,175.384,24.679,154.140
C02923=1081.642,250.954,418.760,175.382,24.676,154.140
C02924=1081.636,250.705,418.788,175.379,24.672,154.139
C02925=1081.631,250.456,418.815,175.377,24.669,154.139
C02926=1081.625,250.208,418.842,175.374,24.665,154.139
C02927=1081.617,249.822,418.884,175.370,24.660,154.138
C02928=1081.607,249.434,418.927,175.366,24.654,154.137
C02929=1081.599,249.047,418.969,175.362,24.649,154.137
C02930=1081.590,248.661,419.012,175.359,24.644,154.136
C02931=1081.585,248.412,419.039,175.356,24.640,154.136
C02932=1081.579,248.163,419.066,175.353,24.637,154.135
C02933=1081.574,247.914,419.094,175.350,24.634,154.135
C02934=1081.568,247.666,419.121,175.348,24.631,154.134
C02935=1081.563,247.418,419.148,175.345,24.627,154.134
C02936=1081.557,247.169,419.175,175.343,24.623,154.134
C02937=1081.552,246.921,419.202,175.340,24.620,154.133
C02938=1081.545,246.672,419.229,175.338,24.617,154.133
C02939=1081.539,246.424,419.256,175.335,24.613,154.132
C02940=1081.534,246.175,419.284,175.333,24.610,154.132
C02941=1081.528,245.927,419.310,175.330,24.606,154.132
C02942=1081.523,245.678,419.337,175.328,24.603,154.131
C02943=1081.518,245.430,419.364,175.325,24.600,154.131
C02944=1081.511,245.181,419.391,175.322,24.597,154.130
C02945=1081.506,244.932,419.418,175.320,24.593,154.130
C02946=1081.500,244.684,419.445,175.317,24.590,154.130
C02947=1081.495,244.435,419.472,175.315,24.587,154.129
C02948=1081.489,244.188,419.499,175.312,24.583,154.129
C02949=1081.483,243.939,419.526,175.310,24.580,154.128
C02950=1081.478,243.691,419.553,175.307,24.576,154.128
C02951=1081.472,243.442,419.580,175.305,24.573,154.128
C02952=1081.466,243.193,419.607,175.302,24.570,154.127
C02953=1081.460,242.945,419.633,175.300,24.566,154.127
C02954=1081.455,242.696,419.661,175.297,24.563,154.126
C02955=1081.449,242.448,419.687,175.294,24.560,154.126
C02956=1081.444,242.199,419.713,175.292,24.557,154.126
C02957=1081.438,241.950,419.740,175.289,24.553,154.125
C02958=1081.432,241.702,419.766,175.287,24.550,154.125
C02959=1081.426,241.454,419.793,175.284,24.546,154.124
C02960=1081.420,241.205,419.820,175.282,24.543,154.124
C02961=1081.414,240.956,419.847,175.279,24.540,154.124
C02962=1081.408,240.708,419.873,175.277,24.536,154.123
C02963=1081.403,240.460,419.900,175.275,24.533,154.123
C02964=1081.398,240.211,419.927,175.271,24.530,154.122
C02965=1081.392,239.962,419.953,175.269,24.527,154.122
C02966=1081.386,239.714,419.980,175.266,24.523,154.122
C02967=1081.381,239.465,420.007,175.264,24.520,154.121
C02968=1081.375,239.217,420.033,175.262,24.517,154.121
C02969=1081.369,238.968,420.060,175.259,24.513,154.120
C02970=1081.364,238.720,420.086,175.257,24.510,154.120
C02971=1081.358,238.471,420.112,175.254,24.506,154.120
C02972=1081.352,238.223,420.139,175.252,24.503,154.119
C02973=1081.346,237.974,420.166,175.249,24.500,154.119
C02974=1081.341,237.725,420.192,175.247,24.496,154.118
C02975=1081.335,237.477,420.218,175.244,24.493,154.118
C02976=1081.329,237.229,420.245,175.241,24.490,154.118
C02977=1081.324,236.980,420.271,175.239,24.486,154.117
C02978=1081.318,236.731,420.298,175.236,24.483,154.117
C02979=1081.308,236.338,420.339,175.233,24.478,154.116
C02980=1081.300,235.944,420.381,175.229,24.472,154.115
C02981=1081.291,235.550,420.422,175.224,24.467,154.115
C02982=1081.282,235.156,420.464,175.221,24.462,154.114
C02983=1081.276,234.907,420.490,175.219,24.459,154.114
C02984=1081.271,234.659,420.517,175.216,24.455,154.114
C02985=1081.265,234.410,420.544,175.214,24.452,154.113
C02986=1081.259,234.161,420.570,175.210,24.449,154.113
C02987=1081.254,233.913,420.596,175.208,24.445,154.112
C02988=1081.247,233.664,420.622,175.206,24.442,154.112
C02989=1081.242,233.416,420.648,175.203,24.439,154.112
C02990=1081.236,233.167,420.674,175.201,24.436,154.111
C02991=1081.231,232.918,420.700,175.199,24.432,154.111
C02992=1081.225,232.670,420.727,175.196,24.429,154.110
C02993=1081.219,232.421,420.753,175.194,24.426,154.110
C02994=1081.214,232.173,420.778,175.191,24.422,154.110
C02995=1081.208,231.924,420.804,175.189,24.419,154.109
C02996=1081.202,231.676,420.831,175.187,24.416,154.109
C02997=1081.197,231.427,420.857,175.183,24.412,154.108
C02998=1081.191,231.178,420.883,175.181,24.409,154.108
C02999=1081.185,230.930,420.909,175.179,24.406,154.108
C03000=1081.179,230.681,420.935,175.176,24.402,154.107
C03001=1081.174,230.432,420.961,175.174,24.399,154.107
C03002=1081.169,230.184,420.987,175.171,24.395,154.106
C03003=1081.163,229.936,421.012,175.169,24.392,154.106
C03004=1081.157,229.687,421.038,175.167,24.389,154.106
C03005=1081.151,229.438,421.065,175.164,24.385,154.105
C03006=1081.145,229.190,421.090,175.162,24.382,154.105
C03007=1081.140,228.941,421.116,175.160,24.379,154.104
C03008=1081.133,228.692,421.141,175.157,24.375,154.104
C03009=1081.128,228.444,421.168,175.154,24.372,154.104
C03010=1081.123,228.195,421.194,175.152,24.369,154.103
C03011=1081.117,227.947,421.219,175.149,24.366,154.103
C03012=1081.111,227.698,421.245,175.147,24.362,154.102
C03013=1081.106,227.449,421.271,175.145,24.359,154.102
C03014=1081.099,227.201,421.297,175.142,24.356,154.102
C03015=1081.094,226.952,421.323,175.140,24.353,154.101
C03016=1081.088,226.704,421.348,175.138,24.350,154.101
C03017=1081.083,226.455,421.374,175.135,24.346,154.101
C03018=1081.076,226.206,421.399,175.132,24.343,154.100
C03019=1081.071,225.957,421.425,175.130,24.340,154.100
C03020=1081.065,225.708,421.451,175.127,24.336,154.099
C03021=1081.060,225.460,421.476,175.125,24.333,154.099
C03022=1081.054,225.211,421.502,175.123,24.330,154.098
C03023=1081.048,224.963,421.527,175.120,24.326,154.098
C03024=1081.043,224.714,421.553,175.118,24.323,154.098
C03025=1081.037,224.466,421.579,175.116,24.320,154.097
C03026=1081.031,224.217,421.605,175.113,24.316,154.097
C03027=1081.025,223.969,421.630,175.111,24.313,154.097
C03028=1081.020,223.720,421.656,175.109,24.310,154.096
C03029=1081.014,223.472,421.681,175.106,24.306,154.096
C03030=1081.009,223.222,421.706,175.103,24.303,154.095
C03031=1081.000,222.820,421.748,175.100,24.297,154.095
C03032=1080.991,222.417,421.789,175.095,24.292,154.094
C03033=1080.981,222.015,421.830,175.092,24.287,154.093
C03034=1080.972,221.613,421.872,175.088,24.282,154.093
C03035=1080.966,221.365,421.897,175.085,24.278,154.092
C03036=1080.961,221.115,421.922,175.083,24.275,154.092
C03037=1080.955,220.867,421.947,175.081,24.272,154.092
C03038=1080.949,220.618,421.972,175.079,24.268,154.091
C03039=1080.944,220.370,421.998,175.076,24.265,154.091
C03040=1080.938,220.121,422.023,175.074,24.262,154.090
C03041=1080.931,219.873,422.049,175.072,24.259,154.090
C03042=1080.927,219.624,422.073,175.069,24.255,154.090
C03043=1080.921,219.375,422.099,175.067,24.252,154.089
C03044=1080.914,219.126,422.124,175.064,24.249,154.089
C03045=1080.910,218.878,422.150,175.062,24.246,154.088
C03046=1080.904,218.629,422.174,175.059,24.242,154.088
C03047=1080.897,218.380,422.200,175.057,24.239,154.088
C03048=1080.892,218.132,422.225,175.055,24.236,154.087
C03049=1080.886,217.883,422.251,175.052,24.232,154.087
C03050=1080.881,217.634,422.275,175.050,24.229,154.086
C03051=1080.875,217.386,422.300,175.048,24.226,154.086
C03052=1080.869,217.137,422.326,175.046,24.222,154.086
C03053=1080.864,216.888,422.350,175.043,24.219,154.085
C03054=1080.858,216.640,422.376,175.041,24.216,154.085
C03055=1080.852,216.390,422.400,175.039,24.212,154.084
C03056=1080.846,216.142,422.425,175.036,24.209,154.084
C03057=1080.841,215.893,422.451,175.033,24.206,154.084
C03058=1080.836,215.645,422.476,175.031,24.202,154.083
C03059=1080.829,215.396,422.501,175.029,24.199,154.083
C03060=1080.824,215.148,422.525,175.026,24.196,154.083
C03061=1080.819,214.899,422.551,175.024,24.192,154.082
C03062=1080.813,214.650,422.575,175.022,24.189,154.082
C03063=1080.807,214.401,422.601,175.020,24.186,154.081
C03064=1080.801,214.153,422.626,175.017,24.182,154.081
C03065=1080.796,213.904,422.650,175.015,24.179,154.080
C03066=1080.790,213.655,422.676,175.013,24.176,154.080
C03067=1080.785,213.406,422.700,175.011,24.173,154.080
C03068=1080.779,213.157,422.725,175.008,24.169,154.079
C03069=1080.773,212.909,422.750,175.006,24.166,154.079
C03070=1080.768,212.660,422.775,175.003,24.163,154.078
C03071=1080.762,212.412,422.800,175.001,24.160,154.078
C03072=1080.756,212.163,422.824,174.998,24.156,154.078
C03073=1080.750,211.915,422.849,174.996,24.153,154.077
C03074=1080.745,211.665,422.874,174.994,24.150,154.077
C03075=1080.739,211.417,422.898,174.992,24.147,154.077
C03076=1080.733,211.168,422.923,174.989,24.143,154.076
C03077=1080.728,210.920,422.948,174.987,24.140,154.076
C03078=1080.722,210.670,422.972,174.985,24.137,154.075
C03079=1080.716,210.422,422.997,174.983,24.134,154.075
C03080=1080.710,210.173,423.022,174.980,24.130,154.075
C03081=1080.705,209.924,423.046,174.977,24.127,154.074
C03082=1080.699,209.676,423.071,174.975,24.124,154.074
C03083=1080.690,209.278,423.111,174.972,24.118,154.073
C03084=1080.681,208.880,423.150,174.968,24.113,154.073
C03085=1080.672,208.481,423.190,174.965,24.108,154.072
C03086=1080.663,208.083,423.229,174.960,24.103,154.071
C03087=1080.639,207.049,423.328,174.863,24.050,154.073
C03088=1080.634,206.801,423.352,174.859,24.047,154.073
C03089=1080.629,206.552,423.377,174.857,24.045,154.073
C03090=1080.622,206.303,423.401,174.854,24.043,154.073
C03091=1080.617,206.054,423.424,174.852,24.040,154.072
C03092=1080.612,205.806,423.449,174.850,24.038,154.072
C03093=1080.606,205.557,423.472,174.847,24.036,154.072
C03094=1080.600,205.307,423.496,174.845,24.034,154.072
C03095=1080.595,205.059,423.520,174.843,24.031,154.072
C03096=1080.589,204.810,423.544,174.840,24.029,154.072
C03097=1080.584,204.562,423.568,174.838,24.027,154.071
C03098=1080.579,204.313,423.592,174.836,24.025,154.071
C03099=1080.573,204.064,423.615,174.833,24.022,154.071
C03100=1080.567,203.815,423.640,174.831,24.020,154.071
C03101=1080.562,203.566,423.664,174.828,24.017,154.071
C03102=1080.556,203.318,423.687,174.826,24.015,154.071
C03103=1080.550,203.069,423.712,174.824,24.013,154.070
C03104=1080.545,202.820,423.735,174.821,24.010,154.070
C03105=1080.539,202.572,423.759,174.818,24.008,154.070
C03106=1080.534,202.322,423.783,174.816,24.006,154.070
C03107=1080.528,202.073,423.806,174.813,24.003,154.070
C03108=1080.522,201.825,423.830,174.811,24.001,154.069
C03109=1080.517,201.576,423.854,174.809,23.998,154.069
C03110=1080.511,201.328,423.877,174.806,23.996,154.069
C03111=1080.506,201.078,423.901,174.804,23.994,154.069
C03112=1080.499,200.829,423.925,174.801,23.992,154.069
C03113=1080.493,200.581,423.948,174.799,23.990,154.069
C03114=1080.488,200.332,423.972,174.797,23.987,154.069
C03115=1080.482,200.083,423.995,174.794,23.985,154.068
C03116=1080.477,199.834,424.019,174.792,23.983,154.068
C03117=1080.471,199.586,424.042,174.790,23.980,154.068
C03118=1080.465,199.337,424.066,174.787,23.978,154.068
C03119=1080.460,199.087,424.090,174.785,23.976,154.068
C03120=1080.454,198.838,424.113,174.782,23.974,154.068
C03121=1080.448,198.590,424.136,174.780,23.972,154.067
C03122=1080.443,198.341,424.160,174.778,23.969,154.067
C03123=1080.437,198.093,424.183,174.775,23.967,154.067
C03124=1080.431,197.844,424.206,174.773,23.964,154.067
C03125=1080.426,197.595,424.230,174.771,23.962,154.067
C03126=1080.420,197.346,424.254,174.768,23.960,154.067
C03127=1080.414,197.097,424.277,174.766,23.958,154.066
C03128=1080.408,196.848,424.301,174.763,23.956,154.066
C03129=1080.403,196.599,424.324,174.761,23.953,154.066
C03130=1080.397,196.350,424.347,174.759,23.951,154.066
C03131=1080.392,196.101,424.371,174.756,23.949,154.066
C03132=1080.386,195.853,424.394,174.754,23.946,154.066
C03133=1080.380,195.604,424.417,174.752,23.944,154.065
C03134=1080.375,195.355,424.441,174.749,23.942,154.065
C03135=1080.369,195.107,424.464,174.747,23.939,154.065
C03136=1080.363,194.858,424.487,174.745,23.937,154.065
C03137=1080.358,194.608,424.511,174.742,23.935,154.065
C03138=1080.353,194.359,424.534,174.740,23.933,154.065
C03139=1080.347,194.111,424.558,174.737,23.930,154.065
C03140=1080.341,193.862,424.580,174.735,23.928,154.064
C03141=1080.336,193.613,424.604,174.733,23.926,154.064
C03142=1080.330,193.364,424.627,174.730,23.923,154.064
C03143=1080.324,193.115,424.650,174.729,23.922,154.064
C03144=1080.318,192.867,424.674,174.726,23.919,154.064
C03145=1080.313,192.618,424.697,174.724,23.917,154.063
C03146=1080.308,192.369,424.720,174.722,23.914,154.063
C03147=1080.302,192.120,424.743,174.719,23.912,154.063
C03148=1080.296,191.841,424.769,174.716,23.910,154.063
C03149=1080.290,191.561,424.795,174.714,23.907,154.063
C03150=1080.284,191.281,424.821,174.711,23.905,154.063
C03151=1080.277,191.001,424.847,174.708,23.902,154.062
C03152=1080.272,190.752,424.870,174.707,23.900,154.062
C03153=1080.266,190.504,424.893,174.704,23.898,154.062
C03154=1080.261,190.254,424.916,174.702,23.895,154.062
C03155=1080.255,190.005,424.939,174.700,23.893,154.062
C03156=1080.250,189.757,424.962,174.697,23.890,154.061
C03157=1080.244,189.508,424.985,174.695,23.888,154.061
C03158=1080.239,189.260,425.008,174.693,23.885,154.061
C03159=1080.234,189.010,425.031,174.690,23.883,154.061
C03160=1080.228,188.761,425.054,174.688,23.881,154.061
C03161=1080.222,188.513,425.077,174.686,23.879,154.061
C03162=1080.217,188.264,425.100,174.683,23.876,154.060
C03163=1080.211,188.015,425.123,174.681,23.874,154.060
C03164=1080.206,187.765,425.147,174.679,23.872,154.060
C03165=1080.201,187.517,425.169,174.677,23.870,154.060
C03166=1080.195,187.268,425.192,174.675,23.867,154.060
C03167=1080.189,187.020,425.215,174.673,23.865,154.059
C03168=1080.183,186.771,425.238,174.670,23.863,154.059
C03169=1080.178,186.521,425.262,174.668,23.860,154.059
C03170=1080.173,186.273,425.285,174.665,23.858,154.059
C03171=1080.168,186.024,425.307,174.663,23.856,154.059
C03172=1080.162,185.775,425.330,174.661,23.853,154.059
C03173=1080.156,185.526,425.352,174.658,23.851,154.058
C03174=1080.151,185.277,425.375,174.656,23.849,154.058
C03175=1080.145,185.028,425.398,174.654,23.846,154.058
C03176=1080.140,184.780,425.421,174.652,23.844,154.058
C03177=1080.134,184.531,425.444,174.650,23.842,154.058
C03178=1080.129,184.282,425.466,174.647,23.840,154.058
C03179=1080.123,184.033,425.489,174.645,23.838,154.057
C03180=1080.116,183.784,425.511,174.643,23.835,154.057
C03181=1080.111,183.535,425.534,174.640,23.833,154.057
C03182=1080.105,183.286,425.557,174.638,23.831,154.057
C03183=1080.100,183.037,425.579,174.636,23.829,154.057
C03184=1080.094,182.788,425.602,174.634,23.827,154.057
C03185=1080.087,182.539,425.625,174.632,23.824,154.056
C03186=1080.083,182.290,425.647,174.629,23.822,154.056
C03187=1080.077,182.042,425.670,174.627,23.820,154.056
C03188=1080.071,181.793,425.693,174.625,23.818,154.056
C03189=1080.065,181.543,425.714,174.622,23.816,154.056
C03190=1080.059,181.295,425.737,174.620,23.813,154.056
C03191=1080.054,181.046,425.760,174.617,23.811,154.056
C03192=1080.048,180.796,425.782,174.616,23.809,154.055
C03193=1080.042,180.548,425.804,174.614,23.807,154.055
C03194=1080.036,180.299,425.827,174.611,23.804,154.055
C03195=1080.031,180.050,425.849,174.609,23.802,154.055
C03196=1080.025,179.801,425.872,174.607,23.800,154.055
C03197=1080.019,179.552,425.894,174.604,23.798,154.055
C03198=1080.014,179.304,425.917,174.602,23.796,154.054
C03199=1080.008,179.055,425.940,174.600,23.794,154.054
C03200=1080.002,178.805,425.961,174.598,23.792,154.054
C03201=1079.996,178.557,425.984,174.596,23.789,154.054
C03202=1079.991,178.307,426.006,174.593,23.787,154.054
C03203=1079.985,178.059,426.028,174.591,23.784,154.054
C03204=1079.980,177.810,426.051,174.589,23.782,154.053
C03205=1079.974,177.561,426.074,174.587,23.780,154.053
C03206=1079.968,177.311,426.095,174.585,23.778,154.053
C03207=1079.963,177.063,426.118,174.582,23.776,154.053
C03208=1079.957,176.814,426.140,174.580,23.774,154.053
C03209=1079.951,176.565,426.162,174.577,23.772,154.053
C03210=1079.945,176.316,426.185,174.575,23.769,154.052
C03211=1079.940,176.067,426.207,174.574,23.767,154.052
C03212=1079.933,175.787,426.232,174.570,23.764,154.052
C03213=1079.927,175.507,426.257,174.568,23.762,154.052
C03214=1079.921,175.227,426.282,174.566,23.759,154.052
C03215=1079.915,174.947,426.306,174.564,23.757,154.052
C03216=1079.909,174.698,426.329,174.561,23.754,154.051
C03217=1079.903,174.449,426.351,174.559,23.752,154.051
C03218=1079.898,174.200,426.373,174.557,23.750,154.051
C03219=1079.892,173.951,426.396,174.555,23.748,154.051
C03220=1079.886,173.702,426.418,174.553,23.746,154.051
C03221=1079.881,173.453,426.439,174.550,23.743,154.051
C03222=1079.876,173.205,426.462,174.548,23.741,154.050
C03223=1079.869,172.955,426.484,174.546,23.739,154.050
C03224=1079.865,172.707,426.506,174.544,23.737,154.050
C03225=1079.858,172.458,426.528,174.542,23.734,154.050
C03226=1079.853,172.208,426.550,174.540,23.732,154.050
C03227=1079.848,171.960,426.572,174.537,23.730,154.050
C03228=1079.842,171.710,426.594,174.535,23.728,154.049
C03229=1079.836,171.461,426.617,174.533,23.726,154.049
C03230=1079.830,171.213,426.638,174.531,23.723,154.049
C03231=1079.825,170.963,426.660,174.529,23.721,154.049
C03232=1079.820,170.715,426.682,174.526,23.719,154.049
C03233=1079.814,170.466,426.705,174.525,23.717,154.048
C03234=1079.808,170.217,426.727,174.523,23.714,154.048
C03235=1079.803,169.968,426.748,174.520,23.712,154.048
C03236=1079.797,169.719,426.770,174.518,23.710,154.048
C03237=1079.792,169.470,426.792,174.515,23.707,154.048
C03238=1079.786,169.221,426.814,174.514,23.705,154.047
C03239=1079.781,168.972,426.836,174.512,23.703,154.047
C03240=1079.775,168.723,426.858,174.509,23.701,154.047
C03241=1079.770,168.474,426.880,174.507,23.698,154.047
C03242=1079.764,168.225,426.902,174.506,23.696,154.047
C03243=1079.759,167.976,426.924,174.503,23.694,154.047
C03244=1079.753,167.727,426.945,174.501,23.692,154.046
C03245=1079.748,167.478,426.967,174.499,23.689,154.046
C03246=1079.742,167.229,426.989,174.496,23.687,154.046
C03247=1079.737,166.980,427.011,174.495,23.685,154.046
C03248=1079.731,166.731,427.032,174.493,23.682,154.046
C03249=1079.725,166.482,427.055,174.490,23.680,154.046
C03250=1079.720,166.234,427.076,174.488,23.678,154.045
C03251=1079.714,165.984,427.098,174.486,23.676,154.045
C03252=1079.709,165.736,427.120,174.484,23.673,154.045
C03253=1079.703,165.486,427.142,174.482,23.671,154.045
C03254=1079.698,165.238,427.163,174.479,23.669,154.045
C03255=1079.693,164.989,427.185,174.478,23.666,154.044
C03256=1079.687,164.740,427.207,174.476,23.664,154.044
C03257=1079.682,164.491,427.229,174.473,23.662,154.044
C03258=1079.676,164.242,427.250,174.472,23.659,154.044
C03259=1079.671,163.992,427.271,174.470,23.657,154.044
C03260=1079.665,163.743,427.293,174.467,23.655,154.043
C03261=1079.660,163.494,427.315,174.465,23.652,154.043
C03262=1079.654,163.245,427.337,174.464,23.650,154.043
C03263=1079.649,162.996,427.358,174.461,23.648,154.043
C03264=1079.644,162.748,427.380,174.459,23.645,154.043
C03265=1079.638,162.498,427.402,174.457,23.643,154.043
C03266=1079.633,162.250,427.423,174.455,23.641,154.042
C03267=1079.627,162.000,427.445,174.453,23.639,154.042
C03268=1079.622,161.752,427.467,174.451,23.636,154.042
C03269=1079.617,161.502,427.488,174.448,23.634,154.042
C03270=1079.611,161.253,427.509,174.447,23.632,154.041
C03271=1079.606,161.004,427.531,174.445,23.630,154.041
C03272=1079.599,160.755,427.552,174.442,23.627,154.041
C03273=1079.594,160.507,427.574,174.441,23.625,154.041
C03274=1079.589,160.257,427.595,174.438,23.623,154.041
C03275=1079.583,160.008,427.616,174.436,23.621,154.041
C03276=1079.577,159.728,427.640,174.434,23.618,154.040
C03277=1079.570,159.447,427.665,174.431,23.616,154.040
C03278=1079.563,159.167,427.689,174.429,23.613,154.040
C03279=1079.557,158.887,427.712,174.427,23.611,154.040
C03280=1079.552,158.638,427.734,174.425,23.608,154.040
C03281=1079.546,158.389,427.756,174.423,23.606,154.039
C03282=1079.541,158.139,427.776,174.421,23.604,154.039
C03283=1079.535,157.890,427.798,174.418,23.602,154.039
C03284=1079.529,157.642,427.819,174.417,23.599,154.039
C03285=1079.524,157.393,427.840,174.415,23.597,154.039
C03286=1079.518,157.143,427.862,174.412,23.595,154.039
C03287=1079.512,156.895,427.883,174.410,23.593,154.038
C03288=1079.507,156.645,427.904,174.409,23.590,154.038
C03289=1079.502,156.396,427.926,174.406,23.588,154.038
C03290=1079.496,156.148,427.947,174.404,23.586,154.038
C03291=1079.490,155.898,427.968,174.403,23.583,154.038
C03292=1079.485,155.649,427.989,174.400,23.581,154.037
C03293=1079.479,155.400,428.010,174.398,23.579,154.037
C03294=1079.473,155.151,428.031,174.396,23.577,154.037
C03295=1079.468,154.903,428.053,174.394,23.574,154.037
C03296=1079.462,154.653,428.073,174.392,23.572,154.037
C03297=1079.456,154.404,428.095,174.390,23.570,154.037
C03298=1079.451,154.155,428.115,174.388,23.568,154.036
C03299=1079.445,153.906,428.137,174.386,23.565,154.036
C03300=1079.440,153.657,428.157,174.384,23.563,154.036
C03301=1079.434,153.408,428.179,174.382,23.561,154.036
C03302=1079.428,153.158,428.200,174.380,23.559,154.036
C03303=1079.423,152.910,428.221,174.378,23.557,154.035
C03304=1079.417,152.661,428.241,174.376,23.554,154.035
C03305=1079.411,152.412,428.263,174.374,23.552,154.035
C03306=1079.406,152.163,428.284,174.372,23.550,154.035
C03307=1079.400,151.914,428.305,174.370,23.548,154.035
C03308=1079.394,151.664,428.326,174.368,23.545,154.035
C03309=1079.389,151.416,428.347,174.366,23.543,154.034
C03310=1079.384,151.167,428.368,174.364,23.541,154.034
C03311=1079.377,150.917,428.389,174.361,23.539,154.034
C03312=1079.372,150.668,428.410,174.360,23.536,154.034
C03313=1079.367,150.419,428.430,174.358,23.534,154.034
C03314=1079.361,150.170,428.452,174.355,23.532,154.033
C03315=1079.356,149.921,428.473,174.354,23.529,154.033
C03316=1079.350,149.672,428.494,174.352,23.527,154.033
C03317=1079.345,149.423,428.514,174.349,23.525,154.033
C03318=1079.339,149.173,428.535,174.348,23.523,154.033
C03319=1079.333,148.925,428.556,174.346,23.520,154.032
C03320=1079.327,148.676,428.577,174.344,23.518,154.032
C03321=1079.321,148.426,428.597,174.342,23.516,154.032
C03322=1079.316,148.178,428.619,174.340,23.513,154.032
C03323=1079.311,147.929,428.639,174.338,23.512,154.032
C03324=1079.305,147.679,428.660,174.336,23.509,154.031
C03325=1079.299,147.430,428.680,174.334,23.507,154.031
C03326=1079.293,147.181,428.701,174.332,23.505,154.031
C03327=1079.288,146.932,428.722,174.330,23.503,154.031
C03328=1079.283,146.683,428.743,174.328,23.500,154.031
C03329=1079.276,146.434,428.764,174.326,23.498,154.030
C03330=1079.271,146.185,428.784,174.324,23.496,154.030
C03331=1079.265,145.936,428.805,174.322,23.493,154.030
C03332=1079.260,145.687,428.825,174.320,23.491,154.030
C03333=1079.253,145.437,428.846,174.318,23.489,154.030
C03334=1079.248,145.189,428.867,174.316,23.487,154.029
C03335=1079.243,144.940,428.887,174.314,23.484,154.029
C03336=1079.237,144.691,428.908,174.313,23.482,154.029
C03337=1079.231,144.441,428.928,174.310,23.480,154.029
C03338=1079.226,144.192,428.949,174.308,23.477,154.029
C03339=1079.220,143.943,428.969,174.307,23.476,154.029
C03340=1079.214,143.663,428.993,174.304,23.473,154.028
C03341=1079.207,143.382,429.016,174.302,23.470,154.028
C03342=1079.201,143.101,429.039,174.300,23.468,154.028
C03343=1079.195,142.821,429.062,174.298,23.465,154.028
C03344=1079.189,142.572,429.082,174.295,23.463,154.028
C03345=1079.184,142.323,429.103,174.294,23.460,154.027
C03346=1079.178,142.073,429.124,174.292,23.458,154.027
C03347=1079.172,141.825,429.144,174.290,23.456,154.027
C03348=1079.166,141.575,429.165,174.288,23.454,154.027
C03349=1079.161,141.326,429.186,174.286,23.451,154.027
C03350=1079.155,141.078,429.206,174.284,23.449,154.026
C03351=1079.150,140.828,429.226,174.282,23.447,154.026
C03352=1079.145,140.579,429.247,174.281,23.444,154.026
C03353=1079.138,140.330,429.267,174.278,23.442,154.026
C03354=1079.133,140.081,429.287,174.276,23.440,154.026
C03355=1079.127,139.831,429.308,174.275,23.438,154.025
C03356=1079.122,139.583,429.328,174.272,23.435,154.025
C03357=1079.116,139.334,429.349,174.271,23.433,154.025
C03358=1079.110,139.085,429.369,174.269,23.431,154.025
C03359=1079.105,138.836,429.389,174.266,23.428,154.025
C03360=1079.098,138.586,429.409,174.265,23.426,154.024
C03361=1079.093,138.337,429.430,174.263,23.424,154.024
C03362=1079.087,138.088,429.449,174.261,23.422,154.024
C03363=1079.082,137.838,429.470,174.259,23.419,154.024
C03364=1079.076,137.590,429.490,174.257,23.417,154.023
C03365=1079.071,137.340,429.510,174.255,23.415,154.023
C03366=1079.065,137.092,429.530,174.253,23.412,154.023
C03367=1079.060,136.843,429.551,174.251,23.411,154.023
C03368=1079.053,136.593,429.571,174.249,23.408,154.023
C03369=1079.048,136.344,429.592,174.248,23.406,154.022
C03370=1079.042,136.095,429.612,174.245,23.404,154.022
C03371=1079.037,135.845,429.631,174.244,23.401,154.022
C03372=1079.031,135.597,429.651,174.242,23.399,154.022
C03373=1079.026,135.347,429.672,174.240,23.397,154.022
C03374=1079.020,135.099,429.692,174.238,23.394,154.021
C03375=1079.014,134.849,429.712,174.236,23.392,154.021
C03376=1079.009,134.600,429.732,174.234,23.390,154.021
C03377=1079.003,134.351,429.752,174.232,23.388,154.021
C03378=1078.997,134.102,429.772,174.231,23.385,154.021
C03379=1078.992,133.853,429.793,174.228,23.383,154.020
C03380=1078.986,133.604,429.813,174.227,23.381,154.020
C03381=1078.981,133.355,429.832,174.225,23.378,154.020
C03382=1078.975,133.106,429.853,174.223,23.376,154.020
C03383=1078.969,132.857,429.873,174.221,23.374,154.020
C03384=1078.964,132.606,429.893,174.219,23.371,154.019
C03385=1078.958,132.358,429.913,174.217,23.369,154.019
C03386=1078.952,132.108,429.933,174.215,23.367,154.019
C03387=1078.946,131.860,429.953,174.214,23.364,154.019
C03388=1078.941,131.610,429.972,174.211,23.362,154.019
C03389=1078.935,131.361,429.992,174.210,23.360,154.018
C03390=1078.929,131.113,430.012,174.208,23.358,154.018
C03391=1078.924,130.863,430.032,174.206,23.356,154.018
C03392=1078.918,130.614,430.052,174.204,23.353,154.018
C03393=1078.912,130.365,430.072,174.203,23.351,154.018
C03394=1078.906,130.116,430.091,174.200,23.349,154.017
C03395=1078.901,129.867,430.112,174.198,23.346,154.017
C03396=1078.895,129.617,430.131,174.197,23.344,154.017
C03397=1078.889,129.368,430.151,174.194,23.342,154.017
C03398=1078.883,129.120,430.171,174.193,23.340,154.017
C03399=1078.878,128.870,430.190,174.191,23.337,154.016
C03400=1078.872,128.621,430.210,174.189,23.335,154.016
C03401=1078.867,128.372,430.230,174.187,23.333,154.016
C03402=1078.861,128.123,430.250,174.186,23.331,154.016
C03403=1078.855,127.873,430.269,174.183,23.328,154.016
C03404=1078.848,127.593,430.292,174.181,23.325,154.015
C03405=1078.842,127.312,430.314,174.180,23.324,154.015
C03406=1078.835,127.031,430.337,174.178,23.321,154.015
C03407=1078.828,126.750,430.358,174.175,23.318,154.015
C03408=1078.822,126.501,430.378,174.173,23.316,154.015
C03409=1078.817,126.252,430.398,174.172,23.313,154.014
C03410=1078.812,126.003,430.418,174.169,23.311,154.014
C03411=1078.806,125.754,430.437,174.168,23.309,154.014
C03412=1078.800,125.505,430.457,174.166,23.306,154.014
C03413=1078.795,125.256,430.476,174.164,23.304,154.013
C03414=1078.789,125.007,430.496,174.162,23.302,154.013
C03415=1078.783,124.757,430.515,174.161,23.299,154.013
C03416=1078.778,124.508,430.535,174.158,23.297,154.013
C03417=1078.772,124.259,430.555,174.157,23.295,154.013
C03418=1078.766,124.009,430.574,174.155,23.293,154.012
C03419=1078.760,123.761,430.594,174.153,23.291,154.012
C03420=1078.755,123.511,430.614,174.151,23.288,154.012
C03421=1078.749,123.262,430.633,174.150,23.286,154.012
C03422=1078.743,123.013,430.653,174.147,23.283,154.011
C03423=1078.737,122.764,430.672,174.146,23.281,154.011
C03424=1078.733,122.515,430.691,174.144,23.279,154.011
C03425=1078.727,122.266,430.711,174.143,23.276,154.011
C03426=1078.721,122.016,430.731,174.140,23.274,154.011
C03427=1078.716,121.767,430.750,174.139,23.272,154.010
C03428=1078.710,121.518,430.770,174.137,23.269,154.010
C03429=1078.704,121.269,430.789,174.135,23.267,154.010
C03430=1078.698,121.019,430.808,174.133,23.265,154.010
C03431=1078.692,120.770,430.828,174.132,23.262,154.009
C03432=1078.687,120.522,430.847,174.129,23.260,154.009
C03433=1078.682,120.272,430.866,174.128,23.258,154.009
C03434=1078.676,120.023,430.886,174.126,23.255,154.009
C03435=1078.670,119.774,430.906,174.124,23.253,154.009
C03436=1078.665,119.524,430.926,174.123,23.251,154.008
C03437=1078.659,119.275,430.945,174.121,23.248,154.008
C03438=1078.654,119.026,430.964,174.119,23.246,154.008
C03439=1078.648,118.777,430.983,174.117,23.244,154.008
C03440=1078.642,118.528,431.003,174.116,23.241,154.007
C03441=1078.637,118.278,431.022,174.114,23.239,154.007
C03442=1078.631,118.029,431.041,174.112,23.237,154.007
C03443=1078.626,117.780,431.060,174.110,23.234,154.007
C03444=1078.620,117.531,431.079,174.109,23.232,154.007
C03445=1078.614,117.282,431.099,174.106,23.229,154.006
C03446=1078.609,117.033,431.119,174.105,23.227,154.006
C03447=1078.604,116.784,431.138,174.103,23.225,154.006
C03448=1078.598,116.534,431.157,174.101,23.222,154.006
C03449=1078.592,116.285,431.176,174.099,23.220,154.005
C03450=1078.586,116.035,431.195,174.098,23.218,154.005
C03451=1078.581,115.787,431.214,174.096,23.215,154.005
C03452=1078.576,115.537,431.233,174.094,23.212,154.005
C03453=1078.570,115.288,431.253,174.093,23.211,154.004
C03454=1078.564,115.039,431.273,174.091,23.208,154.004
C03455=1078.559,114.790,431.291,174.089,23.206,154.004
C03456=1078.553,114.541,431.311,174.087,23.203,154.004
C03457=1078.548,114.291,431.330,174.086,23.201,154.003
C03458=1078.542,114.042,431.349,174.084,23.199,154.003
C03459=1078.537,113.793,431.368,174.082,23.196,154.003
C03460=1078.530,113.544,431.387,174.080,23.194,154.003
C03461=1078.525,113.295,431.406,174.079,23.192,154.003
C03462=1078.519,113.045,431.425,174.076,23.189,154.002
C03463=1078.513,112.796,431.444,174.075,23.187,154.002
C03464=1078.508,112.547,431.463,174.074,23.184,154.002
C03465=1078.502,112.298,431.483,174.071,23.182,154.002
C03466=1078.496,112.049,431.501,174.070,23.180,154.001
C03467=1078.490,111.799,431.520,174.068,23.177,154.001
C03468=1078.485,111.519,431.542,174.066,23.174,154.001
C03469=1078.477,111.238,431.563,174.064,23.172,154.001
C03470=1078.472,110.957,431.584,174.062,23.170,154.000
C03471=1078.465,110.676,431.605,174.060,23.167,154.000
C03472=1078.459,110.427,431.624,174.059,23.164,154.000
C03473=1078.454,110.178,431.643,174.056,23.162,154.000
C03474=1078.447,109.929,431.662,174.055,23.160,154.000
C03475=1078.442,109.679,431.681,174.053,23.158,153.999
C03476=1078.437,109.430,431.700,174.051,23.155,153.999
C03477=1078.430,109.181,431.718,174.050,23.153,153.999
C03478=1078.425,108.931,431.737,174.048,23.150,153.999
C03479=1078.420,108.683,431.756,174.047,23.148,153.998
C03480=1078.413,108.434,431.775,174.044,23.146,153.998
C03481=1078.408,108.184,431.794,174.043,23.143,153.998
C03482=1078.402,107.935,431.813,174.041,23.141,153.998
C03483=1078.396,107.686,431.831,174.039,23.139,153.997
C03484=1078.391,107.436,431.850,174.038,23.136,153.997
C03485=1078.385,107.187,431.869,174.036,23.134,153.997
C03486=1078.379,106.938,431.888,174.034,23.132,153.997
C03487=1078.373,106.689,431.907,174.032,23.129,153.997
C03488=1078.368,106.439,431.926,174.031,23.127,153.996
C03489=1078.362,106.191,431.944,174.029,23.124,153.996
C03490=1078.357,105.941,431.963,174.027,23.122,153.996
C03491=1078.350,105.692,431.982,174.026,23.120,153.996
C03492=1078.345,105.443,432.000,174.024,23.117,153.995
C03493=1078.340,105.193,432.019,174.022,23.115,153.995
C03494=1078.333,104.944,432.038,174.020,23.113,153.995
C03495=1078.328,104.695,432.056,174.019,23.110,153.995
C03496=1078.323,104.445,432.075,174.017,23.107,153.994
C03497=1078.317,104.197,432.093,174.015,23.105,153.994
C03498=1078.312,103.947,432.112,174.014,23.103,153.994
C03499=1078.305,103.698,432.131,174.012,23.100,153.994
C03500=1078.300,103.449,432.150,174.010,23.098,153.993
C03501=1078.295,103.199,432.168,174.008,23.096,153.993
C03502=1078.288,102.950,432.187,174.007,23.093,153.993
C03503=1078.283,102.701,432.206,174.006,23.091,153.993
C03504=1078.277,102.451,432.224,174.003,23.089,153.992
C03505=1078.272,102.203,432.242,174.002,23.086,153.992
C03506=1078.265,101.953,432.261,174.000,23.083,153.992
C03507=1078.261,101.704,432.279,173.998,23.082,153.992
C03508=1078.255,101.455,432.298,173.997,23.079,153.991
C03509=1078.249,101.205,432.316,173.995,23.076,153.991
C03510=1078.244,100.956,432.335,173.994,23.074,153.991
C03511=1078.238,100.706,432.353,173.991,23.072,153.991
C03512=1078.232,100.458,432.371,173.990,23.069,153.990
C03513=1078.226,100.209,432.391,173.989,23.067,153.990
C03514=1078.220,99.959,432.409,173.986,23.065,153.990
C03515=1078.215,99.710,432.428,173.985,23.062,153.990
C03516=1078.209,99.460,432.445,173.983,23.060,153.990
C03517=1078.203,99.212,432.464,173.982,23.058,153.989
C03518=1078.198,98.962,432.482,173.980,23.055,153.989
C03519=1078.191,98.713,432.501,173.978,23.053,153.989
C03520=1078.186,98.464,432.518,173.977,23.050,153.989
C03521=1078.180,98.214,432.538,173.975,23.048,153.988
C03522=1078.174,97.965,432.555,173.973,23.046,153.988
C03523=1078.169,97.716,432.575,173.972,23.043,153.988
C03524=1078.163,97.467,432.592,173.970,23.041,153.988
C03525=1078.157,97.217,432.610,173.968,23.039,153.987
C03526=1078.151,96.968,432.629,173.967,23.036,153.987
C03527=1078.146,96.719,432.647,173.965,23.033,153.987
C03528=1078.140,96.469,432.665,173.963,23.032,153.987
C03529=1078.135,96.220,432.684,173.961,23.029,153.986
C03530=1078.128,95.971,432.702,173.960,23.026,153.986
C03531=1078.123,95.722,432.720,173.959,23.024,153.986
C03532=1078.117,95.441,432.740,173.957,23.021,153.986
C03533=1078.109,95.160,432.761,173.954,23.018,153.985
C03534=1078.104,94.880,432.782,173.953,23.016,153.985
C03535=1078.097,94.599,432.802,173.951,23.013,153.985
C03536=1078.092,94.350,432.820,173.950,23.011,153.985
C03537=1078.085,94.100,432.839,173.947,23.009,153.984
C03538=1078.081,93.851,432.857,173.946,23.006,153.984
C03539=1078.075,93.601,432.875,173.944,23.003,153.984
C03540=1078.069,93.353,432.893,173.943,23.001,153.984
C03541=1078.063,93.103,432.911,173.941,22.999,153.983
C03542=1078.058,92.854,432.929,173.939,22.996,153.983
C03543=1078.051,92.605,432.948,173.938,22.994,153.983
C03544=1078.046,92.356,432.965,173.937,22.991,153.983
C03545=1078.041,92.106,432.984,173.934,22.989,153.982
C03546=1078.035,91.857,433.001,173.933,22.987,153.982
C03547=1078.029,91.608,433.020,173.931,22.984,153.982
C03548=1078.024,91.358,433.038,173.930,22.982,153.982
C03549=1078.018,91.109,433.056,173.928,22.979,153.981
C03550=1078.012,90.859,433.074,173.926,22.977,153.981
C03551=1078.007,90.610,433.091,173.925,22.974,153.981
C03552=1078.000,90.361,433.110,173.923,22.972,153.981
C03553=1077.995,90.112,433.127,173.921,22.969,153.980
C03554=1077.989,89.862,433.145,173.920,22.967,153.980
C03555=1077.983,89.613,433.163,173.919,22.965,153.980
C03556=1077.978,89.363,433.182,173.916,22.962,153.980
C03557=1077.972,89.115,433.200,173.915,22.960,153.979
C03558=1077.966,88.865,433.218,173.913,22.957,153.979
C03559=1077.960,88.616,433.235,173.912,22.955,153.979
C03560=1077.954,88.366,433.253,173.910,22.953,153.979
C03561=1077.949,88.117,433.271,173.908,22.950,153.978
C03562=1077.943,87.868,433.288,173.907,22.948,153.978
C03563=1077.937,87.619,433.306,173.905,22.946,153.978
C03564=1077.931,87.370,433.324,173.903,22.943,153.978
C03565=1077.925,87.120,433.343,173.902,22.941,153.977
C03566=1077.919,86.871,433.360,173.901,22.938,153.977
C03567=1077.913,86.622,433.378,173.898,22.936,153.977
C03568=1077.908,86.373,433.396,173.897,22.933,153.977
C03569=1077.902,86.124,433.413,173.896,22.931,153.976
C03570=1077.896,85.874,433.431,173.894,22.929,153.976
C03571=1077.891,85.625,433.449,173.892,22.926,153.976
C03572=1077.885,85.375,433.467,173.891,22.924,153.976
C03573=1077.880,85.126,433.485,173.889,22.921,153.975
C03574=1077.874,84.877,433.502,173.887,22.919,153.975
C03575=1077.868,84.627,433.520,173.886,22.917,153.975
C03576=1077.863,84.378,433.538,173.884,22.914,153.975
C03577=1077.857,84.129,433.555,173.883,22.911,153.974
C03578=1077.851,83.879,433.573,173.881,22.910,153.974
C03579=1077.845,83.630,433.591,173.879,22.907,153.974
C03580=1077.839,83.380,433.609,173.878,22.904,153.974
C03581=1077.834,83.131,433.626,173.877,22.902,153.973
C03582=1077.828,82.882,433.644,173.875,22.899,153.973
C03583=1077.822,82.632,433.662,173.873,22.897,153.973
C03584=1077.817,82.383,433.679,173.872,22.895,153.972
C03585=1077.811,82.134,433.697,173.870,22.892,153.972
C03586=1077.805,81.885,433.715,173.868,22.890,153.972
C03587=1077.800,81.636,433.733,173.867,22.887,153.972
C03588=1077.794,81.386,433.749,173.865,22.884,153.971
C03589=1077.789,81.137,433.767,173.864,22.882,153.971
C03590=1077.783,80.887,433.785,173.862,22.880,153.971
C03591=1077.777,80.638,433.802,173.860,22.877,153.971
C03592=1077.771,80.389,433.819,173.859,22.875,153.970
C03593=1077.765,80.140,433.837,173.858,22.872,153.970
C03594=1077.759,79.891,433.855,173.856,22.870,153.970
C03595=1077.754,79.641,433.872,173.854,22.867,153.970
C03596=1077.749,79.417,433.889,173.853,22.865,153.969
C03597=1077.744,79.193,433.904,173.852,22.863,153.969
C03598=1077.739,78.968,433.920,173.850,22.861,153.969
C03599=1077.733,78.743,433.936,173.848,22.858,153.969
C03600=1077.729,78.519,433.952,173.847,22.856,153.968
C03601=1077.723,78.294,433.967,173.845,22.854,153.968
C03602=1077.718,78.071,433.983,173.844,22.852,153.968
C03603=1077.713,77.846,433.999,173.843,22.850,153.968
C03604=1077.707,77.596,434.015,173.841,22.847,153.967
C03605=1077.701,77.347,434.033,173.840,22.845,153.967
C03606=1077.695,77.098,434.051,173.838,22.843,153.967
C03607=1077.690,76.849,434.068,173.837,22.840,153.967
C03608=1077.685,76.599,434.085,173.835,22.838,153.966
C03609=1077.678,76.349,434.102,173.833,22.835,153.966
C03610=1077.672,76.100,434.120,173.832,22.832,153.966
C03611=1077.667,75.851,434.137,173.831,22.831,153.966
C03612=1077.661,75.602,434.154,173.828,22.828,153.965
C03613=1077.655,75.352,434.172,173.827,22.825,153.965
C03614=1077.649,75.103,434.189,173.826,22.823,153.965
C03615=1077.644,74.854,434.206,173.824,22.820,153.965
C03616=1077.636,74.524,434.229,173.822,22.817,153.964
C03617=1077.628,74.193,434.252,173.820,22.814,153.964
C03618=1077.621,73.862,434.275,173.818,22.811,153.964
C03619=1077.613,73.532,434.298,173.816,22.807,153.963
C03620=1077.608,73.282,434.315,173.814,22.805,153.963
C03621=1077.602,73.033,434.332,173.812,22.802,153.963
C03622=1077.596,72.783,434.349,173.811,22.800,153.962
C03623=1077.590,72.534,434.367,173.810,22.798,153.962
C03624=1077.584,72.285,434.384,173.808,22.795,153.962
C03625=1077.579,72.036,434.400,173.806,22.792,153.962
C03626=1077.573,71.787,434.418,173.805,22.790,153.961
C03627=1077.567,71.536,434.435,173.804,22.788,153.961
C03628=1077.561,71.288,434.452,173.802,22.785,153.961
C03629=1077.556,71.038,434.469,173.800,22.783,153.961
C03630=1077.550,70.789,434.487,173.799,22.780,153.960
C03631=1077.544,70.540,434.503,173.797,22.778,153.960
C03632=1077.539,70.291,434.520,173.796,22.775,153.960
C03633=1077.533,70.041,434.538,173.794,22.773,153.959
C03634=1077.527,69.791,434.555,173.793,22.770,153.959
C03635=1077.521,69.542,434.572,173.791,22.768,153.959
C03636=1077.516,69.293,434.589,173.790,22.765,153.959
C03637=1077.510,69.044,434.606,173.788,22.763,153.958
C03638=1077.504,68.794,434.623,173.786,22.760,153.958
